RoboDK station: kr30 cnc 072119 dry run.rdk

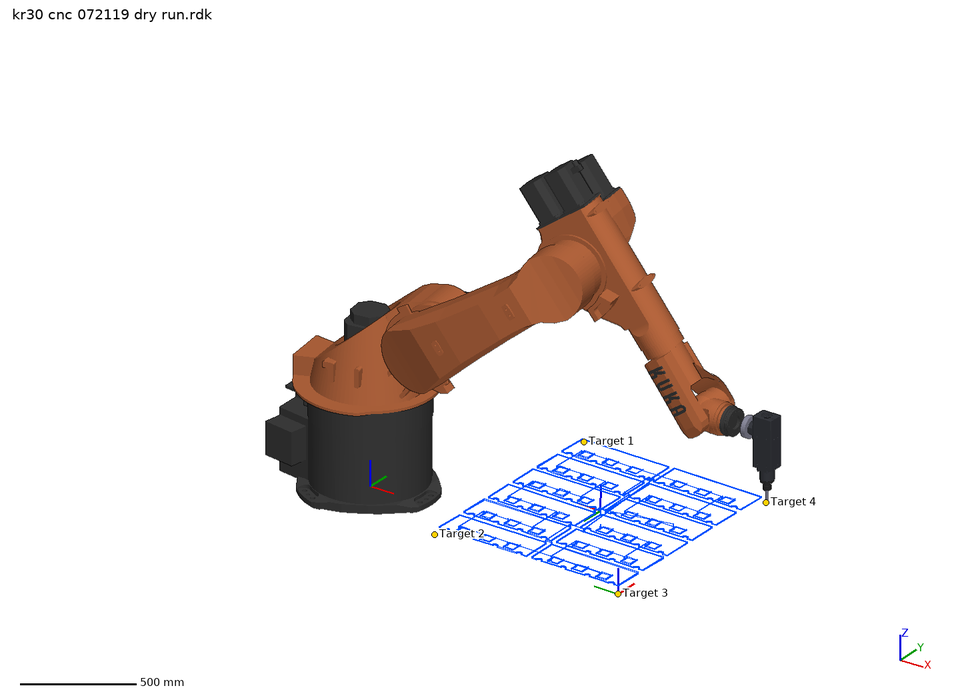
[picture v0: the station drawn from its stored meshes, robots at their saved joint values, targets as dots, program paths as lines]
Station kr30 cnc 072119 dry run. Poses are relative to the parent item; angles as X-Y-Z fixed-axis rotations.
  - frame GIGASHEEN Base at (0, 0, 0) mm
    - robot GIGASHEEN (model KUKA KR 30 HA): 6 axes, payload 30 kg, reach 2033 mm, repeatability 0.05 mm, weight 665 kg
        modified DH rows (alpha deg, a mm, theta deg, d mm): 0, 0, 0, 815; -90, 350, 0, 0; 0, 850, -90, 0; -90, 145, 0, 820; 90, 0, 0, 0; -90, 0, 180, 170
        joint limits [-185, -135, -120, -350, -119, -350] to [185, 35, 158, 350, 119, 350]; home [0, -90, 90, 0, 0, 0]; saved at [-6.898, -35.989, 90.741, -8.88, -55.221, 5.167]
      - tool 1/2" End Mill TCP, TCP at (337.71, -2.2, 160.57) mm, rotated rx 0 ry 90 rz 0 deg, size 415.8 x 102 x 153.6 mm
    - target Target 1 (joint target) at (982.46, 202.21, 406.25) mm, rotated rx -179.95 ry 0.15 rz -89.48 deg; joints [7.49, -59.642, 144.935, 97.969, -90.801, -4.608] of GIGASHEEN
    - target Target 2 (joint target) at (986.83, -921.64, 412.07) mm, rotated rx -179.94 ry 0.15 rz -89.48 deg; joints [51.766, -38.608, 94.384, 136.851, -116.554, -22.567] of GIGASHEEN
    - target Target 3 (joint target) at (1949.02, -919.97, 396.91) mm, rotated rx -179.94 ry 0.14 rz 179.61 deg; joints [29.5, -22.76, 62.288, 41.088, -47.759, -30.404] of GIGASHEEN
    - target Target 4 (joint target) at (1949.02, 190.94, 391.63) mm, rotated rx -179.94 ry 0.14 rz 179.61 deg; joints [-6.898, -35.989, 90.741, -8.88, -55.221, 5.167] of GIGASHEEN
  - machining project Machining Settings: C:/Users/liqui/OneDrive/Desktop/first half pipe jig.apt | rotZ(0) | rotX(0)*rotY(0) | rotZ(0)
  - program Machining (1954 instructions, listed below)
  - program Prog2 (4 instructions, listed below)
  - frame Table at (1949.02, -919.97, 396.91) mm, rotated rx 0.87 ry 0.27 rz 90 deg
    - frame Frame 4 at (550, 480, 40) mm, rotated rx 0 ry 0 rz 90 deg
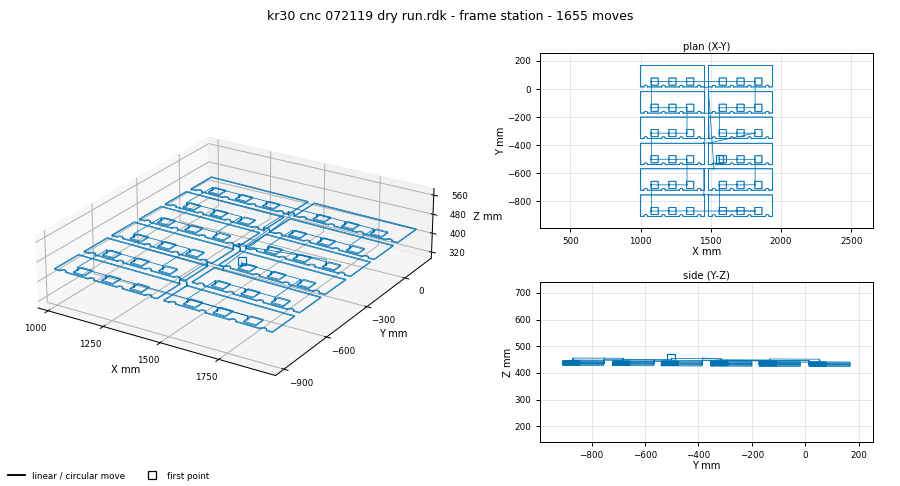
[picture p0: tool path of kr30 cnc 072119 dry run.rdk in frame station, 1655 of 1659 moves have a stored position in this frame; points joined in program order, loops and branches not executed]

--- program Machining (robot GIGASHEEN) ---
  Smooth(0)
  Set Ref.: Frame 4
  Set Tool: 1/2" End Mill TCP
  Show 1/2" End Mill TCP
  Print: /'1001'
  Print: /''
  Print: /'2D Contour2'
  Set speed (500.0 mm/s)
  MoveJ 1 to (-92.16, 131.48, 15) mm, rotated rx 180 ry 0 rz 0 deg; joints [21.909, -52.477, 118.543, 23.9, -67.031, -9.189]
  MoveL 2 to (-92.16, 131.48, 15) mm, rotated rx 180 ry 0 rz 0 deg; joints [21.909, -52.477, 118.543, 23.9, -67.031, -9.189]
  MoveL 3 to (-92.16, 131.48, 15) mm, rotated rx 180 ry 0 rz 0 deg; joints [21.909, -52.477, 118.543, 23.9, -67.031, -9.189]
  Set speed (500.0 mm/s)
  MoveL 4 to (-92.16, 131.48, 6) mm, rotated rx -180 ry 0 rz 0 deg; joints [21.913, -51.95, 118.536, 23.816, -67.508, -8.962]
  Set speed (25.4 mm/s)
  MoveL 5 to (-92.16, 131.48, -3.54) mm, rotated rx 180 ry 0 rz 0 deg; joints [21.917, -51.387, 118.521, 23.73, -68.011, -8.725]
  MoveC 6 to (-91.98, 131.48, -3.99) mm, rotated rx 180 ry 0 rz 0 deg; joints [21.92, -51.367, 118.535, 23.728, -68.042, -8.712] to (-91.53, 131.48, -4.17) mm, rotated rx -180 ry 0 rz 0 deg; joints [21.927, -51.372, 118.57, 23.731, -68.07, -8.702]
  Set speed (50.8 mm/s)
  MoveL 7 to (-90.89, 131.48, -4.18) mm, rotated rx 180 ry 0 rz 0 deg; joints [21.937, -51.395, 118.619, 23.737, -68.095, -8.694]
  MoveC 8 to (-90.44, 131.3, -4.18) mm, rotated rx 180 ry 0 rz 0 deg; joints [21.937, -51.415, 118.66, 23.734, -68.115, -8.685] to (-90.26, 130.85, -4.18) mm, rotated rx -180 ry 0 rz 0 deg; joints [21.922, -51.428, 118.688, 23.715, -68.127, -8.672]
  MoveL 9 to (-90.26, 105.45, -4.17) mm, rotated rx -180 ry 0 rz 0 deg; joints [20.901, -51.776, 119.463, 22.561, -68.365, -8.105]
  MoveL 10 to (-141.06, 105.45, -4.17) mm, rotated rx 180 ry 0 rz 0 deg; joints [20.142, -49.88, 115.443, 22.086, -66.286, -8.677]
  MoveL 11 to (-141.06, 156.25, -4.18) mm, rotated rx 180 ry 0 rz 0 deg; joints [22.112, -49.164, 113.869, 24.362, -65.824, -9.881]
  MoveL 12 to (-90.26, 156.25, -4.18) mm, rotated rx -180 ry 0 rz 0 deg; joints [22.93, -51.06, 117.875, 24.862, -67.882, -9.257]
  MoveL 13 to (-90.26, 130.85, -4.18) mm, rotated rx -180 ry 0 rz 0 deg; joints [21.922, -51.428, 118.688, 23.715, -68.127, -8.672]
  MoveC 14 to (-90.44, 130.4, -4.17) mm, rotated rx 180 ry 0 rz 0 deg; joints [21.901, -51.427, 118.688, 23.693, -68.123, -8.664] to (-90.89, 130.21, -4.18) mm, rotated rx -180 ry 0 rz 0 deg; joints [21.887, -51.413, 118.659, 23.68, -68.107, -8.665]
  MoveL 15 to (-91.53, 130.21, -4.18) mm, rotated rx -180 ry 0 rz 0 deg; joints [21.877, -51.39, 118.609, 23.673, -68.082, -8.673]
  MoveC 16 to (-91.98, 130.21, -3.99) mm, rotated rx 180 ry 0 rz 0 deg; joints [21.869, -51.385, 118.575, 23.67, -68.054, -8.683] to (-92.16, 130.21, -3.54) mm, rotated rx 180 ry 0 rz 0 deg; joints [21.866, -51.404, 118.561, 23.672, -68.023, -8.696]
  Set speed (500.0 mm/s)
  MoveL 17 to (-92.16, 130.21, 5) mm, rotated rx 180 ry 0 rz 0 deg; joints [21.862, -51.909, 118.575, 23.749, -67.573, -8.908]
  MoveL 18 to (-92.16, 131.49, 5) mm, rotated rx -180 ry 0 rz 0 deg; joints [21.913, -51.891, 118.535, 23.807, -67.561, -8.937]
  Set speed (25.4 mm/s)
  MoveL 19 to (-92.16, 131.48, 1.82) mm, rotated rx 180 ry 0 rz 0 deg; joints [21.914, -51.704, 118.531, 23.778, -67.729, -8.858]
  MoveL 20 to (-92.16, 131.48, -7.72) mm, rotated rx 180 ry 0 rz 0 deg; joints [21.919, -51.139, 118.513, 23.693, -68.23, -8.622]
  MoveC 21 to (-91.98, 131.48, -8.16) mm, rotated rx 180 ry 0 rz 0 deg; joints [21.922, -51.119, 118.526, 23.691, -68.261, -8.609] to (-91.53, 131.48, -8.35) mm, rotated rx -180 ry 0 rz 0 deg; joints [21.929, -51.124, 118.56, 23.694, -68.288, -8.599]
  Set speed (50.8 mm/s)
  MoveL 22 to (-90.89, 131.48, -8.35) mm, rotated rx 180 ry 0 rz 0 deg; joints [21.939, -51.148, 118.61, 23.701, -68.314, -8.591]
  MoveC 23 to (-90.44, 131.3, -8.35) mm, rotated rx 180 ry 0 rz 0 deg; joints [21.939, -51.167, 118.651, 23.697, -68.334, -8.582] to (-90.26, 130.85, -8.35) mm, rotated rx -180 ry 0 rz 0 deg; joints [21.924, -51.18, 118.679, 23.679, -68.346, -8.57]
  MoveL 24 to (-90.26, 105.45, -8.35) mm, rotated rx -180 ry 0 rz 0 deg; joints [20.902, -51.526, 119.454, 22.526, -68.588, -8.006]
  MoveL 25 to (-141.06, 105.45, -8.35) mm, rotated rx -180 ry 0 rz 0 deg; joints [20.144, -49.641, 115.434, 22.05, -66.499, -8.584]
  MoveL 26 to (-141.06, 156.25, -8.35) mm, rotated rx 180 ry 0 rz 0 deg; joints [22.114, -48.93, 113.86, 24.322, -66.03, -9.779]
  MoveL 27 to (-90.26, 156.25, -8.35) mm, rotated rx -180 ry 0 rz 0 deg; joints [22.931, -50.815, 117.866, 24.823, -68.097, -9.15]
  MoveL 28 to (-90.26, 130.85, -8.35) mm, rotated rx -180 ry 0 rz 0 deg; joints [21.924, -51.18, 118.679, 23.679, -68.346, -8.57]
  MoveC 29 to (-90.44, 130.4, -8.35) mm, rotated rx 180 ry 0 rz 0 deg; joints [21.903, -51.179, 118.679, 23.657, -68.343, -8.562] to (-90.89, 130.21, -8.35) mm, rotated rx -180 ry 0 rz 0 deg; joints [21.889, -51.165, 118.65, 23.644, -68.326, -8.563]
  MoveL 30 to (-91.53, 130.21, -8.35) mm, rotated rx 180 ry 0 rz 0 deg; joints [21.878, -51.142, 118.6, 23.637, -68.301, -8.57]
  MoveC 31 to (-91.98, 130.21, -8.16) mm, rotated rx -180 ry 0 rz 0 deg; joints [21.871, -51.137, 118.566, 23.634, -68.273, -8.58] to (-92.16, 130.21, -7.72) mm, rotated rx -180 ry 0 rz 0 deg; joints [21.868, -51.157, 118.552, 23.636, -68.242, -8.593]
  Set speed (500.0 mm/s)
  MoveL 32 to (-92.16, 130.21, 6) mm, rotated rx 180 ry 0 rz 0 deg; joints [21.862, -51.968, 118.576, 23.758, -67.52, -8.933]
  MoveL 33 to (-219.16, 131.48, 6) mm, rotated rx -180 ry 0 rz 0 deg; joints [20.042, -46.998, 108.236, 22.771, -62.271, -10.462]
  Set speed (25.4 mm/s)
  MoveL 34 to (-219.16, 131.48, -3.54) mm, rotated rx -180 ry 0 rz 0 deg; joints [20.045, -46.495, 108.222, 22.677, -62.723, -10.251]
  MoveC 35 to (-218.98, 131.48, -3.99) mm, rotated rx -180 ry 0 rz 0 deg; joints [20.048, -46.478, 108.237, 22.673, -62.752, -10.239] to (-218.53, 131.48, -4.17) mm, rotated rx -180 ry 0 rz 0 deg; joints [20.054, -46.487, 108.275, 22.674, -62.78, -10.229]
  Set speed (50.8 mm/s)
  MoveL 36 to (-217.89, 131.49, -4.17) mm, rotated rx -180 ry 0 rz 0 deg; joints [20.063, -46.512, 108.328, 22.678, -62.808, -10.221]
  MoveC 37 to (-217.44, 131.3, -4.18) mm, rotated rx 180 ry 0 rz 0 deg; joints [20.062, -46.533, 108.372, 22.673, -62.829, -10.211] to (-217.26, 130.85, -4.18) mm, rotated rx -180 ry 0 rz 0 deg; joints [20.048, -46.547, 108.402, 22.654, -62.841, -10.197]
  MoveL 38 to (-217.26, 105.45, -4.17) mm, rotated rx 180 ry 0 rz 0 deg; joints [19.099, -46.897, 109.164, 21.526, -63.055, -9.56]
  MoveL 39 to (-268.06, 105.45, -4.17) mm, rotated rx -180 ry 0 rz 0 deg; joints [18.46, -44.806, 104.789, 21.257, -60.816, -10.178]
  MoveL 40 to (-268.06, 156.25, -4.18) mm, rotated rx -180 ry 0 rz 0 deg; joints [20.293, -44.079, 103.221, 23.503, -60.392, -11.532]
  MoveL 41 to (-217.26, 156.25, -4.18) mm, rotated rx -180 ry 0 rz 0 deg; joints [20.986, -46.177, 107.599, 23.778, -62.618, -10.849]
  MoveL 42 to (-217.26, 130.85, -4.18) mm, rotated rx -180 ry 0 rz 0 deg; joints [20.048, -46.547, 108.402, 22.654, -62.841, -10.197]
  MoveC 43 to (-217.44, 130.4, -4.17) mm, rotated rx -180 ry 0 rz 0 deg; joints [20.029, -46.546, 108.4, 22.633, -62.836, -10.188] to (-217.89, 130.21, -4.18) mm, rotated rx -180 ry 0 rz 0 deg; joints [20.016, -46.53, 108.368, 22.622, -62.819, -10.189]
  MoveL 44 to (-218.53, 130.21, -4.18) mm, rotated rx -180 ry 0 rz 0 deg; joints [20.007, -46.505, 108.314, 22.618, -62.791, -10.197]
  MoveC 45 to (-218.98, 130.21, -3.99) mm, rotated rx 180 ry 0 rz 0 deg; joints [20.001, -46.496, 108.276, 22.617, -62.763, -10.206] to (-219.16, 130.21, -3.54) mm, rotated rx -180 ry 0 rz 0 deg; joints [19.998, -46.513, 108.261, 22.62, -62.734, -10.218]
  Set speed (500.0 mm/s)
  MoveL 46 to (-219.16, 130.21, 5) mm, rotated rx -180 ry 0 rz 0 deg; joints [19.995, -46.963, 108.274, 22.704, -62.329, -10.407]
  MoveL 47 to (-219.16, 131.48, 5) mm, rotated rx 180 ry 0 rz 0 deg; joints [20.042, -46.945, 108.235, 22.761, -62.319, -10.44]
  Set speed (25.4 mm/s)
  MoveL 48 to (-219.16, 131.48, 1.82) mm, rotated rx -180 ry 0 rz 0 deg; joints [20.043, -46.778, 108.231, 22.729, -62.469, -10.369]
  MoveL 49 to (-219.16, 131.48, -7.72) mm, rotated rx -180 ry 0 rz 0 deg; joints [20.047, -46.273, 108.214, 22.636, -62.919, -10.159]
  MoveC 50 to (-218.98, 131.48, -8.16) mm, rotated rx -180 ry 0 rz 0 deg; joints [20.05, -46.257, 108.228, 22.633, -62.949, -10.147] to (-218.53, 131.48, -8.35) mm, rotated rx -180 ry 0 rz 0 deg; joints [20.056, -46.265, 108.266, 22.634, -62.977, -10.138]
  Set speed (50.8 mm/s)
  MoveL 51 to (-217.89, 131.48, -8.35) mm, rotated rx -180 ry 0 rz 0 deg; joints [20.064, -46.291, 108.32, 22.638, -63.004, -10.13]
  MoveC 52 to (-217.44, 131.3, -8.35) mm, rotated rx -180 ry 0 rz 0 deg; joints [20.064, -46.311, 108.363, 22.633, -63.025, -10.119] to (-217.26, 130.85, -8.35) mm, rotated rx 180 ry 0 rz 0 deg; joints [20.05, -46.325, 108.393, 22.614, -63.037, -10.106]
  MoveL 53 to (-217.26, 105.45, -8.35) mm, rotated rx -180 ry 0 rz 0 deg; joints [19.101, -46.674, 109.156, 21.488, -63.255, -9.473]
  MoveL 54 to (-268.06, 105.45, -8.35) mm, rotated rx -180 ry 0 rz 0 deg; joints [18.461, -44.592, 104.78, 21.217, -61.008, -10.094]
  MoveL 55 to (-268.06, 156.25, -8.35) mm, rotated rx -180 ry 0 rz 0 deg; joints [20.295, -43.868, 103.212, 23.459, -60.578, -11.44]
  MoveL 56 to (-217.26, 156.25, -8.35) mm, rotated rx 180 ry 0 rz 0 deg; joints [20.987, -45.957, 107.59, 23.736, -62.812, -10.754]
  MoveL 57 to (-217.26, 130.85, -8.35) mm, rotated rx 180 ry 0 rz 0 deg; joints [20.05, -46.325, 108.393, 22.614, -63.037, -10.106]
  MoveC 58 to (-217.44, 130.4, -8.35) mm, rotated rx 180 ry 0 rz 0 deg; joints [20.03, -46.324, 108.391, 22.593, -63.033, -10.097] to (-217.89, 130.21, -8.35) mm, rotated rx -180 ry 0 rz 0 deg; joints [20.017, -46.309, 108.359, 22.582, -63.015, -10.098]
  MoveL 59 to (-218.53, 130.21, -8.35) mm, rotated rx -180 ry 0 rz 0 deg; joints [20.009, -46.283, 108.305, 22.578, -62.988, -10.106]
  MoveC 60 to (-218.98, 130.21, -8.16) mm, rotated rx 180 ry 0 rz 0 deg; joints [20.003, -46.275, 108.267, 22.577, -62.96, -10.115] to (-219.16, 130.22, -7.72) mm, rotated rx -180 ry 0 rz 0 deg; joints [20, -46.291, 108.253, 22.58, -62.93, -10.127]
  Set speed (500.0 mm/s)
  MoveL 61 to (-219.16, 130.21, 6) mm, rotated rx -180 ry 0 rz 0 deg; joints [19.995, -47.016, 108.276, 22.714, -62.282, -10.429]
  MoveL 62 to (-346.16, 131.48, 6) mm, rotated rx -180 ry 0 rz 0 deg; joints [18.455, -41.516, 96.931, 22.283, -56.572, -12.158]
  Set speed (25.4 mm/s)
  MoveL 63 to (-346.16, 131.48, -3.54) mm, rotated rx 180 ry 0 rz 0 deg; joints [18.458, -41.062, 96.917, 22.178, -56.98, -11.961]
  MoveC 64 to (-345.98, 131.48, -3.99) mm, rotated rx -180 ry 0 rz 0 deg; joints [18.461, -41.049, 96.933, 22.173, -57.008, -11.95] to (-345.53, 131.48, -4.17) mm, rotated rx -180 ry 0 rz 0 deg; joints [18.466, -41.06, 96.975, 22.172, -57.037, -11.939]
  Set speed (50.8 mm/s)
  MoveL 65 to (-344.89, 131.48, -4.17) mm, rotated rx -180 ry 0 rz 0 deg; joints [18.473, -41.089, 97.035, 22.173, -57.067, -11.93]
  MoveC 66 to (-344.44, 131.3, -4.17) mm, rotated rx 180 ry 0 rz 0 deg; joints [18.472, -41.112, 97.083, 22.165, -57.09, -11.918] to (-344.26, 130.85, -4.18) mm, rotated rx -180 ry 0 rz 0 deg; joints [18.459, -41.127, 97.114, 22.146, -57.103, -11.902]
  MoveL 67 to (-344.26, 105.45, -4.17) mm, rotated rx -180 ry 0 rz 0 deg; joints [17.574, -41.489, 97.887, 21.018, -57.305, -11.178]
  MoveL 68 to (-395.06, 105.45, -4.18) mm, rotated rx -180 ry 0 rz 0 deg; joints [17.029, -39.137, 93.017, 20.982, -54.842, -11.914]
  MoveL 69 to (-395.06, 156.25, -4.17) mm, rotated rx -180 ry 0 rz 0 deg; joints [18.741, -38.377, 91.402, 23.257, -54.433, -13.468]
  MoveL 70 to (-344.26, 156.25, -4.18) mm, rotated rx 180 ry 0 rz 0 deg; joints [19.334, -40.745, 96.299, 23.273, -56.893, -12.643]
  MoveL 71 to (-344.26, 130.85, -4.18) mm, rotated rx -180 ry 0 rz 0 deg; joints [18.459, -41.127, 97.114, 22.146, -57.103, -11.902]
  MoveC 72 to (-344.44, 130.4, -4.18) mm, rotated rx -180 ry 0 rz 0 deg; joints [18.441, -41.125, 97.111, 22.125, -57.097, -11.892] to (-344.89, 130.22, -4.18) mm, rotated rx -180 ry 0 rz 0 deg; joints [18.429, -41.108, 97.074, 22.116, -57.078, -11.893]
  MoveL 73 to (-345.53, 130.21, -4.18) mm, rotated rx 180 ry 0 rz 0 deg; joints [18.422, -41.079, 97.015, 22.115, -57.048, -11.902]
  MoveC 74 to (-345.98, 130.21, -3.99) mm, rotated rx -180 ry 0 rz 0 deg; joints [18.417, -41.068, 96.973, 22.117, -57.018, -11.913] to (-346.16, 130.21, -3.54) mm, rotated rx 180 ry 0 rz 0 deg; joints [18.414, -41.081, 96.956, 22.121, -56.99, -11.925]
  Set speed (500.0 mm/s)
  MoveL 75 to (-346.16, 130.21, 5) mm, rotated rx -180 ry 0 rz 0 deg; joints [18.411, -41.488, 96.969, 22.215, -56.625, -12.101]
  MoveL 76 to (-346.16, 131.48, 5) mm, rotated rx -180 ry 0 rz 0 deg; joints [18.455, -41.469, 96.93, 22.272, -56.615, -12.138]
  Set speed (25.4 mm/s)
  MoveL 77 to (-346.16, 131.48, 1.82) mm, rotated rx -180 ry 0 rz 0 deg; joints [18.456, -41.318, 96.926, 22.236, -56.751, -12.072]
  MoveL 78 to (-346.16, 131.48, -7.72) mm, rotated rx -180 ry 0 rz 0 deg; joints [18.46, -40.862, 96.908, 22.133, -57.158, -11.876]
  MoveC 79 to (-345.98, 131.48, -8.16) mm, rotated rx 180 ry 0 rz 0 deg; joints [18.462, -40.849, 96.925, 22.128, -57.186, -11.865] to (-345.53, 131.48, -8.35) mm, rotated rx -180 ry 0 rz 0 deg; joints [18.467, -40.86, 96.966, 22.127, -57.215, -11.854]
  Set speed (50.8 mm/s)
  MoveL 80 to (-344.89, 131.48, -8.35) mm, rotated rx -180 ry 0 rz 0 deg; joints [18.475, -40.889, 97.026, 22.128, -57.245, -11.845]
  MoveC 81 to (-344.44, 131.3, -8.35) mm, rotated rx 180 ry 0 rz 0 deg; joints [18.473, -40.912, 97.074, 22.12, -57.268, -11.833] to (-344.26, 130.85, -8.35) mm, rotated rx -180 ry 0 rz 0 deg; joints [18.46, -40.927, 97.105, 22.101, -57.28, -11.817]
  MoveL 82 to (-344.26, 105.45, -8.35) mm, rotated rx 180 ry 0 rz 0 deg; joints [17.576, -41.287, 97.879, 20.976, -57.485, -11.097]
  MoveL 83 to (-395.06, 105.45, -8.35) mm, rotated rx -180 ry 0 rz 0 deg; joints [17.03, -38.943, 93.009, 20.937, -55.015, -11.834]
  MoveL 84 to (-395.06, 156.25, -8.35) mm, rotated rx -180 ry 0 rz 0 deg; joints [18.742, -38.186, 91.393, 23.207, -54.602, -13.38]
  MoveL 85 to (-344.26, 156.25, -8.35) mm, rotated rx -180 ry 0 rz 0 deg; joints [19.335, -40.546, 96.29, 23.226, -57.068, -12.555]
  MoveL 86 to (-344.26, 130.85, -8.35) mm, rotated rx -180 ry 0 rz 0 deg; joints [18.46, -40.927, 97.105, 22.101, -57.28, -11.817]
  MoveC 87 to (-344.44, 130.4, -8.35) mm, rotated rx -180 ry 0 rz 0 deg; joints [18.442, -40.925, 97.102, 22.081, -57.275, -11.807] to (-344.89, 130.21, -8.35) mm, rotated rx -180 ry 0 rz 0 deg; joints [18.431, -40.908, 97.066, 22.072, -57.255, -11.808]
  MoveL 88 to (-345.53, 130.21, -8.35) mm, rotated rx -180 ry 0 rz 0 deg; joints [18.423, -40.879, 97.006, 22.071, -57.225, -11.818]
  MoveC 89 to (-345.98, 130.21, -8.16) mm, rotated rx -180 ry 0 rz 0 deg; joints [18.418, -40.868, 96.964, 22.072, -57.196, -11.828] to (-346.16, 130.21, -7.72) mm, rotated rx 180 ry 0 rz 0 deg; joints [18.416, -40.881, 96.948, 22.076, -57.168, -11.84]
  Set speed (500.0 mm/s)
  MoveL 90 to (-346.16, 130.21, 6) mm, rotated rx -180 ry 0 rz 0 deg; joints [18.411, -41.535, 96.971, 22.226, -56.582, -12.121]
  MoveL 91 to (-346.16, 313.35, 6) mm, rotated rx 180 ry 0 rz 0 deg; joints [24.501, -38.28, 90.113, 30.424, -54.956, -17.966]
  Set speed (25.4 mm/s)
  MoveL 92 to (-346.16, 313.35, -3.54) mm, rotated rx 180 ry 0 rz 0 deg; joints [24.504, -37.849, 90.099, 30.281, -55.317, -17.711]
  MoveC 93 to (-345.98, 313.35, -3.99) mm, rotated rx -180 ry 0 rz 0 deg; joints [24.507, -37.837, 90.116, 30.275, -55.343, -17.695] to (-345.53, 313.35, -4.17) mm, rotated rx -180 ry 0 rz 0 deg; joints [24.514, -37.85, 90.159, 30.272, -55.371, -17.681]
  Set speed (50.8 mm/s)
  MoveL 94 to (-344.89, 313.36, -4.18) mm, rotated rx -180 ry 0 rz 0 deg; joints [24.523, -37.879, 90.22, 30.271, -55.401, -17.668]
  MoveC 95 to (-344.44, 313.17, -4.18) mm, rotated rx -180 ry 0 rz 0 deg; joints [24.524, -37.904, 90.271, 30.263, -55.424, -17.652] to (-344.26, 312.72, -4.18) mm, rotated rx -180 ry 0 rz 0 deg; joints [24.512, -37.922, 90.309, 30.243, -55.438, -17.633]
  MoveL 96 to (-344.26, 287.32, -4.18) mm, rotated rx -180 ry 0 rz 0 deg; joints [23.697, -38.438, 91.398, 29.106, -55.691, -16.768]
  MoveL 97 to (-395.06, 287.32, -4.18) mm, rotated rx 180 ry 0 rz 0 deg; joints [22.998, -36.008, 86.396, 29.181, -53.234, -17.841]
  MoveL 98 to (-395.06, 338.12, -4.18) mm, rotated rx 180 ry 0 rz 0 deg; joints [24.581, -34.921, 84.111, 31.512, -52.717, -19.704]
  MoveL 99 to (-344.26, 338.12, -4.18) mm, rotated rx 180 ry 0 rz 0 deg; joints [25.316, -37.384, 89.172, 31.383, -55.178, -18.521]
  MoveL 100 to (-344.26, 312.72, -4.17) mm, rotated rx 180 ry 0 rz 0 deg; joints [24.512, -37.922, 90.309, 30.243, -55.438, -17.633]
  MoveC 101 to (-344.44, 312.27, -4.17) mm, rotated rx -180 ry 0 rz 0 deg; joints [24.495, -37.923, 90.31, 30.223, -55.433, -17.621] to (-344.89, 312.08, -4.17) mm, rotated rx -180 ry 0 rz 0 deg; joints [24.483, -37.906, 90.275, 30.214, -55.414, -17.624]
  MoveL 102 to (-345.53, 312.08, -4.18) mm, rotated rx 180 ry 0 rz 0 deg; joints [24.473, -37.876, 90.214, 30.215, -55.384, -17.637]
  MoveC 103 to (-345.98, 312.08, -3.99) mm, rotated rx 180 ry 0 rz 0 deg; joints [24.467, -37.864, 90.171, 30.218, -55.356, -17.652] to (-346.16, 312.08, -3.54) mm, rotated rx 180 ry 0 rz 0 deg; joints [24.464, -37.875, 90.154, 30.224, -55.33, -17.667]
  Set speed (500.0 mm/s)
  MoveL 104 to (-346.16, 312.08, 5) mm, rotated rx -180 ry 0 rz 0 deg; joints [24.461, -38.262, 90.167, 30.352, -55.007, -17.895]
  MoveL 105 to (-346.16, 313.35, 5) mm, rotated rx -180 ry 0 rz 0 deg; joints [24.501, -38.235, 90.112, 30.409, -54.994, -17.939]
  Set speed (25.4 mm/s)
  MoveL 106 to (-346.16, 313.35, 1.82) mm, rotated rx -180 ry 0 rz 0 deg; joints [24.502, -38.092, 90.108, 30.361, -55.115, -17.854]
  MoveL 107 to (-346.16, 313.35, -7.71) mm, rotated rx -180 ry 0 rz 0 deg; joints [24.506, -37.659, 90.09, 30.22, -55.474, -17.601]
  MoveC 108 to (-345.98, 313.35, -8.16) mm, rotated rx 180 ry 0 rz 0 deg; joints [24.509, -37.647, 90.107, 30.213, -55.5, -17.586] to (-345.53, 313.35, -8.35) mm, rotated rx -180 ry 0 rz 0 deg; joints [24.515, -37.66, 90.15, 30.211, -55.528, -17.571]
  Set speed (50.8 mm/s)
  MoveL 109 to (-344.89, 313.35, -8.35) mm, rotated rx 180 ry 0 rz 0 deg; joints [24.525, -37.689, 90.211, 30.21, -55.558, -17.558]
  MoveC 110 to (-344.44, 313.17, -8.35) mm, rotated rx -180 ry 0 rz 0 deg; joints [24.525, -37.714, 90.262, 30.202, -55.582, -17.542] to (-344.26, 312.72, -8.35) mm, rotated rx -180 ry 0 rz 0 deg; joints [24.514, -37.732, 90.3, 30.182, -55.595, -17.523]
  MoveL 111 to (-344.26, 287.32, -8.35) mm, rotated rx -180 ry 0 rz 0 deg; joints [23.699, -38.246, 91.389, 29.047, -55.852, -16.661]
  MoveL 112 to (-395.06, 287.32, -8.35) mm, rotated rx 180 ry 0 rz 0 deg; joints [22.999, -35.823, 86.387, 29.119, -53.388, -17.735]
  MoveL 113 to (-395.06, 338.12, -8.35) mm, rotated rx -180 ry 0 rz 0 deg; joints [24.583, -34.738, 84.102, 31.445, -52.865, -19.591]
  MoveL 114 to (-344.26, 338.12, -8.35) mm, rotated rx 180 ry 0 rz 0 deg; joints [25.318, -37.195, 89.164, 31.32, -55.332, -18.408]
  MoveL 115 to (-344.26, 312.72, -8.35) mm, rotated rx -180 ry 0 rz 0 deg; joints [24.514, -37.732, 90.3, 30.182, -55.595, -17.523]
  MoveC 116 to (-344.44, 312.27, -8.35) mm, rotated rx 180 ry 0 rz 0 deg; joints [24.497, -37.733, 90.302, 30.162, -55.591, -17.511] to (-344.89, 312.08, -8.35) mm, rotated rx -180 ry 0 rz 0 deg; joints [24.484, -37.716, 90.267, 30.153, -55.571, -17.514]
  MoveL 117 to (-345.53, 312.08, -8.35) mm, rotated rx 180 ry 0 rz 0 deg; joints [24.475, -37.686, 90.205, 30.154, -55.541, -17.528]
  MoveC 118 to (-345.98, 312.08, -8.16) mm, rotated rx 180 ry 0 rz 0 deg; joints [24.468, -37.674, 90.163, 30.157, -55.513, -17.542] to (-346.16, 312.08, -7.72) mm, rotated rx 180 ry 0 rz 0 deg; joints [24.465, -37.685, 90.146, 30.163, -55.487, -17.558]
  Set speed (500.0 mm/s)
  MoveL 119 to (-346.16, 312.08, 6) mm, rotated rx 180 ry 0 rz 0 deg; joints [24.46, -38.307, 90.168, 30.367, -54.969, -17.921]
  MoveL 120 to (-219.16, 313.35, 6) mm, rotated rx -180 ry 0 rz 0 deg; joints [26.482, -43.877, 101.587, 30.778, -60.597, -15.594]
  Set speed (25.4 mm/s)
  MoveL 121 to (-219.16, 313.35, -3.54) mm, rotated rx 180 ry 0 rz 0 deg; joints [26.486, -43.405, 101.574, 30.651, -60.993, -15.327]
  MoveC 122 to (-218.98, 313.35, -3.99) mm, rotated rx -180 ry 0 rz 0 deg; joints [26.489, -43.39, 101.589, 30.646, -61.019, -15.312] to (-218.53, 313.35, -4.17) mm, rotated rx -180 ry 0 rz 0 deg; joints [26.496, -43.399, 101.626, 30.647, -61.046, -15.299]
  Set speed (50.8 mm/s)
  MoveL 123 to (-217.89, 313.35, -4.17) mm, rotated rx -180 ry 0 rz 0 deg; joints [26.507, -43.425, 101.68, 30.65, -61.073, -15.288]
  MoveC 124 to (-217.44, 313.17, -4.17) mm, rotated rx -180 ry 0 rz 0 deg; joints [26.508, -43.448, 101.726, 30.645, -61.094, -15.275] to (-217.26, 312.72, -4.18) mm, rotated rx -180 ry 0 rz 0 deg; joints [26.496, -43.464, 101.761, 30.627, -61.106, -15.258]
  MoveL 125 to (-217.26, 287.32, -4.18) mm, rotated rx 180 ry 0 rz 0 deg; joints [25.634, -43.956, 102.815, 29.523, -61.366, -14.493]
  MoveL 126 to (-268.06, 287.32, -4.18) mm, rotated rx 180 ry 0 rz 0 deg; joints [24.825, -41.833, 98.411, 29.263, -59.167, -15.349]
  MoveL 127 to (-268.06, 338.12, -4.17) mm, rotated rx -180 ry 0 rz 0 deg; joints [26.499, -40.813, 96.241, 31.488, -58.649, -16.97]
  MoveL 128 to (-217.26, 338.12, -4.17) mm, rotated rx -180 ry 0 rz 0 deg; joints [27.346, -42.951, 100.666, 31.729, -60.841, -16.044]
  MoveL 129 to (-217.26, 312.72, -4.18) mm, rotated rx -180 ry 0 rz 0 deg; joints [26.496, -43.464, 101.761, 30.627, -61.106, -15.258]
  MoveC 130 to (-217.44, 312.27, -4.17) mm, rotated rx 180 ry 0 rz 0 deg; joints [26.478, -43.465, 101.764, 30.606, -61.103, -15.248] to (-217.89, 312.08, -4.18) mm, rotated rx -180 ry 0 rz 0 deg; joints [26.464, -43.451, 101.734, 30.595, -61.086, -15.25]
  MoveL 131 to (-218.53, 312.08, -4.17) mm, rotated rx -180 ry 0 rz 0 deg; joints [26.454, -43.425, 101.68, 30.591, -61.059, -15.26]
  MoveC 132 to (-218.98, 312.08, -3.99) mm, rotated rx -180 ry 0 rz 0 deg; joints [26.446, -43.415, 101.642, 30.591, -61.032, -15.273] to (-219.16, 312.08, -3.54) mm, rotated rx -180 ry 0 rz 0 deg; joints [26.443, -43.43, 101.627, 30.596, -61.006, -15.289]
  Set speed (500.0 mm/s)
  MoveL 133 to (-219.16, 312.08, 5) mm, rotated rx 180 ry 0 rz 0 deg; joints [26.439, -43.853, 101.64, 30.709, -60.652, -15.526]
  MoveL 134 to (-219.16, 313.35, 5) mm, rotated rx 180 ry 0 rz 0 deg; joints [26.482, -43.828, 101.586, 30.764, -60.639, -15.566]
  Set speed (25.4 mm/s)
  MoveL 135 to (-219.16, 313.35, 1.82) mm, rotated rx -180 ry 0 rz 0 deg; joints [26.483, -43.671, 101.582, 30.722, -60.771, -15.477]
  MoveL 136 to (-219.16, 313.36, -7.72) mm, rotated rx -180 ry 0 rz 0 deg; joints [26.487, -43.197, 101.565, 30.597, -61.165, -15.212]
  MoveC 137 to (-218.98, 313.35, -8.16) mm, rotated rx 180 ry 0 rz 0 deg; joints [26.491, -43.182, 101.58, 30.592, -61.191, -15.197] to (-218.53, 313.36, -8.35) mm, rotated rx -180 ry 0 rz 0 deg; joints [26.498, -43.191, 101.618, 30.593, -61.218, -15.184]
  Set speed (50.8 mm/s)
  MoveL 138 to (-217.89, 313.35, -8.35) mm, rotated rx 180 ry 0 rz 0 deg; joints [26.509, -43.217, 101.672, 30.596, -61.245, -15.173]
  MoveC 139 to (-217.44, 313.17, -8.35) mm, rotated rx -180 ry 0 rz 0 deg; joints [26.51, -43.239, 101.718, 30.591, -61.266, -15.16] to (-217.26, 312.72, -8.35) mm, rotated rx 180 ry 0 rz 0 deg; joints [26.498, -43.256, 101.753, 30.573, -61.278, -15.143]
  MoveL 140 to (-217.26, 287.32, -8.35) mm, rotated rx -180 ry 0 rz 0 deg; joints [25.636, -43.746, 102.806, 29.471, -61.542, -14.381]
  MoveL 141 to (-268.06, 287.32, -8.35) mm, rotated rx -180 ry 0 rz 0 deg; joints [24.826, -41.63, 98.402, 29.208, -59.337, -15.239]
  MoveL 142 to (-268.06, 338.12, -8.35) mm, rotated rx 180 ry 0 rz 0 deg; joints [26.501, -40.614, 96.233, 31.43, -58.812, -16.855]
  MoveL 143 to (-217.26, 338.12, -8.35) mm, rotated rx -180 ry 0 rz 0 deg; joints [27.348, -42.745, 100.657, 31.673, -61.009, -15.926]
  MoveL 144 to (-217.26, 312.72, -8.35) mm, rotated rx 180 ry 0 rz 0 deg; joints [26.498, -43.256, 101.753, 30.573, -61.278, -15.143]
  MoveC 145 to (-217.44, 312.27, -8.35) mm, rotated rx -180 ry 0 rz 0 deg; joints [26.48, -43.257, 101.756, 30.552, -61.275, -15.133] to (-217.89, 312.08, -8.35) mm, rotated rx -180 ry 0 rz 0 deg; joints [26.466, -43.242, 101.725, 30.541, -61.258, -15.135]
  MoveL 146 to (-218.53, 312.08, -8.35) mm, rotated rx -180 ry 0 rz 0 deg; joints [26.455, -43.216, 101.671, 30.537, -61.231, -15.145]
  MoveC 147 to (-218.98, 312.08, -8.16) mm, rotated rx 180 ry 0 rz 0 deg; joints [26.448, -43.207, 101.634, 30.537, -61.204, -15.158] to (-219.16, 312.08, -7.72) mm, rotated rx -180 ry 0 rz 0 deg; joints [26.445, -43.222, 101.619, 30.542, -61.178, -15.174]
  Set speed (500.0 mm/s)
  MoveL 148 to (-219.16, 312.08, 6) mm, rotated rx -180 ry 0 rz 0 deg; joints [26.439, -43.903, 101.641, 30.722, -60.61, -15.554]
  MoveL 149 to (-92.16, 313.35, 6) mm, rotated rx -180 ry 0 rz 0 deg; joints [28.782, -48.856, 111.85, 31.879, -65.703, -13.605]
  Set speed (25.4 mm/s)
  MoveL 150 to (-92.16, 313.35, -3.54) mm, rotated rx 180 ry 0 rz 0 deg; joints [28.786, -48.334, 111.836, 31.764, -66.135, -13.313]
  MoveC 151 to (-91.98, 313.35, -3.99) mm, rotated rx -180 ry 0 rz 0 deg; joints [28.79, -48.316, 111.85, 31.761, -66.163, -13.297] to (-91.53, 313.35, -4.17) mm, rotated rx -180 ry 0 rz 0 deg; joints [28.799, -48.322, 111.884, 31.764, -66.189, -13.285]
  Set speed (50.8 mm/s)
  MoveL 152 to (-90.89, 313.35, -4.18) mm, rotated rx -180 ry 0 rz 0 deg; joints [28.811, -48.346, 111.933, 31.771, -66.213, -13.275]
  MoveC 153 to (-90.44, 313.17, -4.18) mm, rotated rx -180 ry 0 rz 0 deg; joints [28.813, -48.366, 111.975, 31.769, -66.233, -13.263] to (-90.26, 312.72, -4.18) mm, rotated rx -180 ry 0 rz 0 deg; joints [28.801, -48.381, 112.008, 31.751, -66.245, -13.248]
  MoveL 154 to (-90.26, 287.32, -4.17) mm, rotated rx -180 ry 0 rz 0 deg; joints [27.888, -48.865, 113.06, 30.652, -66.523, -12.552]
  MoveL 155 to (-141.06, 287.32, -4.18) mm, rotated rx 180 ry 0 rz 0 deg; joints [26.944, -46.965, 109.081, 30.121, -64.514, -13.303]
  MoveL 156 to (-141.06, 338.12, -4.18) mm, rotated rx -180 ry 0 rz 0 deg; joints [28.715, -45.973, 106.942, 32.313, -63.97, -14.764]
  MoveL 157 to (-90.26, 338.12, -4.17) mm, rotated rx 180 ry 0 rz 0 deg; joints [29.698, -47.878, 110.917, 32.843, -65.963, -13.964]
  MoveL 158 to (-90.26, 312.72, -4.18) mm, rotated rx -180 ry 0 rz 0 deg; joints [28.801, -48.381, 112.008, 31.751, -66.245, -13.248]
  MoveC 159 to (-90.44, 312.27, -4.18) mm, rotated rx 180 ry 0 rz 0 deg; joints [28.781, -48.383, 112.013, 31.73, -66.243, -13.238] to (-90.89, 312.08, -4.17) mm, rotated rx 180 ry 0 rz 0 deg; joints [28.766, -48.37, 111.986, 31.717, -66.227, -13.24]
  MoveL 160 to (-91.53, 312.08, -4.18) mm, rotated rx -180 ry 0 rz 0 deg; joints [28.753, -48.347, 111.937, 31.709, -66.203, -13.249]
  MoveC 161 to (-91.98, 312.08, -3.99) mm, rotated rx -180 ry 0 rz 0 deg; joints [28.745, -48.341, 111.903, 31.706, -66.177, -13.262] to (-92.16, 312.08, -3.54) mm, rotated rx -180 ry 0 rz 0 deg; joints [28.741, -48.358, 111.89, 31.71, -66.149, -13.278]
  Set speed (500.0 mm/s)
  MoveL 162 to (-92.16, 312.08, 5) mm, rotated rx 180 ry 0 rz 0 deg; joints [28.737, -48.826, 111.903, 31.812, -65.762, -13.538]
  MoveL 163 to (-92.16, 313.36, 5) mm, rotated rx -180 ry 0 rz 0 deg; joints [28.782, -48.801, 111.849, 31.867, -65.748, -13.574]
  Set speed (25.4 mm/s)
  MoveL 164 to (-92.16, 313.35, 1.83) mm, rotated rx -180 ry 0 rz 0 deg; joints [28.783, -48.628, 111.845, 31.829, -65.892, -13.477]
  MoveL 165 to (-92.16, 313.35, -7.71) mm, rotated rx 180 ry 0 rz 0 deg; joints [28.788, -48.104, 111.828, 31.715, -66.324, -13.187]
  MoveC 166 to (-91.98, 313.35, -8.16) mm, rotated rx 180 ry 0 rz 0 deg; joints [28.792, -48.086, 111.841, 31.712, -66.351, -13.171] to (-91.53, 313.35, -8.35) mm, rotated rx -180 ry 0 rz 0 deg; joints [28.801, -48.093, 111.875, 31.715, -66.377, -13.158]
  Set speed (50.8 mm/s)
  MoveL 167 to (-90.89, 313.35, -8.35) mm, rotated rx 180 ry 0 rz 0 deg; joints [28.813, -48.116, 111.924, 31.722, -66.402, -13.149]
  MoveC 168 to (-90.44, 313.17, -8.35) mm, rotated rx -180 ry 0 rz 0 deg; joints [28.815, -48.136, 111.966, 31.72, -66.421, -13.137] to (-90.26, 312.72, -8.35) mm, rotated rx -180 ry 0 rz 0 deg; joints [28.803, -48.151, 111.999, 31.702, -66.433, -13.122]
  MoveL 169 to (-90.26, 287.32, -8.35) mm, rotated rx 180 ry 0 rz 0 deg; joints [27.89, -48.633, 113.052, 30.605, -66.716, -12.428]
  MoveL 170 to (-141.06, 287.32, -8.35) mm, rotated rx 180 ry 0 rz 0 deg; joints [26.946, -46.741, 109.072, 30.072, -64.7, -13.185]
  MoveL 171 to (-141.06, 338.12, -8.35) mm, rotated rx -180 ry 0 rz 0 deg; joints [28.716, -45.754, 106.933, 32.261, -64.148, -14.64]
  MoveL 172 to (-90.26, 338.12, -8.35) mm, rotated rx -180 ry 0 rz 0 deg; joints [29.7, -47.65, 110.908, 32.793, -66.147, -13.835]
  MoveL 173 to (-90.26, 312.72, -8.35) mm, rotated rx -180 ry 0 rz 0 deg; joints [28.803, -48.151, 111.999, 31.702, -66.433, -13.122]
  MoveC 174 to (-90.44, 312.27, -8.35) mm, rotated rx -180 ry 0 rz 0 deg; joints [28.783, -48.153, 112.004, 31.681, -66.431, -13.112] to (-90.89, 312.08, -8.35) mm, rotated rx 180 ry 0 rz 0 deg; joints [28.768, -48.14, 111.977, 31.668, -66.416, -13.114]
  MoveL 175 to (-91.53, 312.08, -8.35) mm, rotated rx -180 ry 0 rz 0 deg; joints [28.755, -48.117, 111.929, 31.66, -66.391, -13.123]
  MoveC 176 to (-91.98, 312.08, -8.16) mm, rotated rx -180 ry 0 rz 0 deg; joints [28.747, -48.111, 111.895, 31.658, -66.365, -13.136] to (-92.16, 312.08, -7.72) mm, rotated rx -180 ry 0 rz 0 deg; joints [28.743, -48.129, 111.881, 31.661, -66.338, -13.152]
  Set speed (500.0 mm/s)
  MoveL 177 to (-92.16, 312.08, 6) mm, rotated rx -180 ry 0 rz 0 deg; joints [28.736, -48.881, 111.904, 31.824, -65.716, -13.569]
  MoveL 178 to (-92.16, 499.69, 6) mm, rotated rx 180 ry 0 rz 0 deg; joints [34.993, -44.649, 102.911, 39.778, -63.653, -19.397]
  Set speed (25.4 mm/s)
  MoveL 179 to (-92.16, 499.69, -3.54) mm, rotated rx 180 ry 0 rz 0 deg; joints [34.998, -44.171, 102.898, 39.637, -64.012, -19.069]
  MoveC 180 to (-91.98, 499.69, -3.99) mm, rotated rx 180 ry 0 rz 0 deg; joints [35.002, -44.155, 102.911, 39.633, -64.036, -19.05] to (-91.53, 499.69, -4.17) mm, rotated rx -180 ry 0 rz 0 deg; joints [35.012, -44.162, 102.946, 39.635, -64.06, -19.035]
  Set speed (50.8 mm/s)
  MoveL 181 to (-90.89, 499.69, -4.18) mm, rotated rx 180 ry 0 rz 0 deg; joints [35.026, -44.186, 102.995, 39.641, -64.084, -19.024]
  MoveC 182 to (-90.44, 499.51, -4.17) mm, rotated rx -180 ry 0 rz 0 deg; joints [35.03, -44.208, 103.039, 39.638, -64.103, -19.009] to (-90.26, 499.06, -4.18) mm, rotated rx 180 ry 0 rz 0 deg; joints [35.02, -44.226, 103.078, 39.622, -64.115, -18.99]
  MoveL 183 to (-90.26, 473.66, -4.18) mm, rotated rx 180 ry 0 rz 0 deg; joints [34.221, -44.857, 104.424, 38.566, -64.412, -18.138]
  MoveL 184 to (-141.06, 473.66, -4.17) mm, rotated rx -180 ry 0 rz 0 deg; joints [33.155, -42.929, 100.434, 38.077, -62.45, -19.078]
  MoveL 185 to (-141.06, 524.46, -4.18) mm, rotated rx -180 ry 0 rz 0 deg; joints [34.714, -41.63, 97.681, 40.216, -61.861, -20.866]
  MoveL 186 to (-90.26, 524.46, -4.17) mm, rotated rx -180 ry 0 rz 0 deg; joints [35.803, -43.573, 101.689, 40.674, -63.816, -19.867]
  MoveL 187 to (-90.26, 499.06, -4.18) mm, rotated rx 180 ry 0 rz 0 deg; joints [35.02, -44.226, 103.078, 39.622, -64.115, -18.99]
  MoveC 188 to (-90.44, 498.61, -4.17) mm, rotated rx -180 ry 0 rz 0 deg; joints [35.002, -44.23, 103.087, 39.601, -64.113, -18.978] to (-90.89, 498.42, -4.17) mm, rotated rx -180 ry 0 rz 0 deg; joints [34.986, -44.218, 103.063, 39.589, -64.098, -18.98]
  MoveL 189 to (-91.53, 498.42, -4.17) mm, rotated rx -180 ry 0 rz 0 deg; joints [34.972, -44.195, 103.014, 39.582, -64.074, -18.992]
  MoveC 190 to (-91.98, 498.42, -3.99) mm, rotated rx -180 ry 0 rz 0 deg; joints [34.963, -44.187, 102.98, 39.58, -64.05, -19.007] to (-92.16, 498.42, -3.54) mm, rotated rx -180 ry 0 rz 0 deg; joints [34.958, -44.203, 102.966, 39.584, -64.027, -19.026]
  Set speed (500.0 mm/s)
  MoveL 191 to (-92.16, 498.42, 5) mm, rotated rx -180 ry 0 rz 0 deg; joints [34.954, -44.631, 102.979, 39.71, -63.705, -19.319]
  MoveL 192 to (-92.16, 499.69, 5) mm, rotated rx -180 ry 0 rz 0 deg; joints [34.994, -44.599, 102.91, 39.763, -63.691, -19.363]
  Set speed (25.4 mm/s)
  MoveL 193 to (-92.16, 499.69, 1.83) mm, rotated rx -180 ry 0 rz 0 deg; joints [34.995, -44.44, 102.906, 39.716, -63.81, -19.253]
  MoveL 194 to (-92.16, 499.69, -7.72) mm, rotated rx 180 ry 0 rz 0 deg; joints [35, -43.961, 102.89, 39.577, -64.168, -18.927]
  MoveC 195 to (-91.98, 499.69, -8.16) mm, rotated rx -180 ry 0 rz 0 deg; joints [35.004, -43.945, 102.903, 39.572, -64.192, -18.908] to (-91.53, 499.69, -8.35) mm, rotated rx 180 ry 0 rz 0 deg; joints [35.014, -43.952, 102.937, 39.574, -64.216, -18.893]
  Set speed (50.8 mm/s)
  MoveL 196 to (-90.89, 499.69, -8.35) mm, rotated rx 180 ry 0 rz 0 deg; joints [35.028, -43.976, 102.986, 39.581, -64.24, -18.881]
  MoveC 197 to (-90.44, 499.51, -8.35) mm, rotated rx -180 ry 0 rz 0 deg; joints [35.032, -43.997, 103.031, 39.578, -64.259, -18.867] to (-90.26, 499.06, -8.35) mm, rotated rx -180 ry 0 rz 0 deg; joints [35.022, -44.015, 103.069, 39.561, -64.271, -18.848]
  MoveL 198 to (-90.26, 473.66, -8.35) mm, rotated rx -180 ry 0 rz 0 deg; joints [34.223, -44.644, 104.415, 38.507, -64.573, -17.997]
  MoveL 199 to (-141.06, 473.66, -8.35) mm, rotated rx -180 ry 0 rz 0 deg; joints [33.157, -42.723, 100.426, 38.016, -62.606, -18.942]
  MoveL 200 to (-141.06, 524.46, -8.35) mm, rotated rx -180 ry 0 rz 0 deg; joints [34.716, -41.429, 97.673, 40.152, -62.009, -20.726]
  MoveL 201 to (-90.26, 524.46, -8.35) mm, rotated rx -180 ry 0 rz 0 deg; joints [35.805, -43.365, 101.681, 40.612, -63.968, -19.723]
  MoveL 202 to (-90.26, 499.06, -8.35) mm, rotated rx -180 ry 0 rz 0 deg; joints [35.022, -44.015, 103.069, 39.561, -64.271, -18.848]
  MoveC 203 to (-90.44, 498.61, -8.35) mm, rotated rx -180 ry 0 rz 0 deg; joints [35.004, -44.02, 103.079, 39.541, -64.27, -18.836] to (-90.89, 498.42, -8.35) mm, rotated rx 180 ry 0 rz 0 deg; joints [34.988, -44.008, 103.055, 39.528, -64.255, -18.838]
  MoveL 204 to (-91.53, 498.42, -8.35) mm, rotated rx -180 ry 0 rz 0 deg; joints [34.974, -43.984, 103.006, 39.522, -64.231, -18.85]
  MoveC 205 to (-91.98, 498.42, -8.16) mm, rotated rx 180 ry 0 rz 0 deg; joints [34.965, -43.977, 102.972, 39.52, -64.207, -18.865] to (-92.16, 498.42, -7.72) mm, rotated rx -180 ry 0 rz 0 deg; joints [34.96, -43.993, 102.958, 39.524, -64.183, -18.883]
  Set speed (500.0 mm/s)
  MoveL 206 to (-92.16, 498.42, 6) mm, rotated rx 180 ry 0 rz 0 deg; joints [34.954, -44.681, 102.98, 39.725, -63.667, -19.354]
  MoveL 207 to (-219.16, 499.69, 6) mm, rotated rx 180 ry 0 rz 0 deg; joints [32.409, -39.564, 92.515, 38.877, -58.619, -21.95]
  Set speed (25.4 mm/s)
  MoveL 208 to (-219.16, 499.69, -3.54) mm, rotated rx -180 ry 0 rz 0 deg; joints [32.413, -39.126, 92.502, 38.72, -58.951, -21.641]
  MoveC 209 to (-218.98, 499.69, -3.99) mm, rotated rx -180 ry 0 rz 0 deg; joints [32.417, -39.113, 92.517, 38.713, -58.975, -21.622] to (-218.53, 499.69, -4.17) mm, rotated rx -180 ry 0 rz 0 deg; joints [32.426, -39.123, 92.556, 38.712, -59, -21.606]
  Set speed (50.8 mm/s)
  MoveL 210 to (-217.89, 499.69, -4.18) mm, rotated rx 180 ry 0 rz 0 deg; joints [32.438, -39.15, 92.611, 38.715, -59.027, -21.592]
  MoveC 211 to (-217.44, 499.51, -4.18) mm, rotated rx -180 ry 0 rz 0 deg; joints [32.441, -39.174, 92.66, 38.708, -59.048, -21.575] to (-217.26, 499.06, -4.18) mm, rotated rx 180 ry 0 rz 0 deg; joints [32.431, -39.194, 92.702, 38.689, -59.061, -21.554]
  MoveL 212 to (-217.26, 473.66, -4.18) mm, rotated rx -180 ry 0 rz 0 deg; joints [31.663, -39.848, 94.081, 37.59, -59.352, -20.618]
  MoveL 213 to (-268.06, 473.66, -4.18) mm, rotated rx -180 ry 0 rz 0 deg; joints [30.733, -37.649, 89.56, 37.447, -57.17, -21.76]
  MoveL 214 to (-268.06, 524.46, -4.17) mm, rotated rx -180 ry 0 rz 0 deg; joints [32.232, -36.283, 86.693, 39.705, -56.582, -23.755]
  MoveL 215 to (-217.26, 524.46, -4.17) mm, rotated rx -180 ry 0 rz 0 deg; joints [33.186, -38.515, 91.273, 39.791, -58.767, -22.518]
  MoveL 216 to (-217.26, 499.06, -4.18) mm, rotated rx 180 ry 0 rz 0 deg; joints [32.431, -39.194, 92.702, 38.689, -59.061, -21.554]
  MoveC 217 to (-217.44, 498.61, -4.18) mm, rotated rx 180 ry 0 rz 0 deg; joints [32.414, -39.198, 92.71, 38.669, -59.058, -21.542] to (-217.89, 498.42, -4.17) mm, rotated rx 180 ry 0 rz 0 deg; joints [32.4, -39.183, 92.681, 38.66, -59.042, -21.545]
  MoveL 218 to (-218.53, 498.42, -4.17) mm, rotated rx 180 ry 0 rz 0 deg; joints [32.387, -39.157, 92.626, 38.657, -59.015, -21.559]
  MoveC 219 to (-218.98, 498.42, -3.99) mm, rotated rx 180 ry 0 rz 0 deg; joints [32.379, -39.146, 92.587, 38.658, -58.989, -21.575] to (-219.16, 498.42, -3.54) mm, rotated rx 180 ry 0 rz 0 deg; joints [32.375, -39.159, 92.572, 38.665, -58.966, -21.593]
  Set speed (500.0 mm/s)
  MoveL 220 to (-219.16, 498.42, 5) mm, rotated rx -180 ry 0 rz 0 deg; joints [32.371, -39.552, 92.584, 38.805, -58.668, -21.87]
  MoveL 221 to (-219.16, 499.69, 5) mm, rotated rx -180 ry 0 rz 0 deg; joints [32.41, -39.518, 92.514, 38.86, -58.654, -21.917]
  Set speed (25.4 mm/s)
  MoveL 222 to (-219.16, 499.69, 1.82) mm, rotated rx 180 ry 0 rz 0 deg; joints [32.411, -39.373, 92.51, 38.808, -58.765, -21.814]
  MoveL 223 to (-219.16, 499.69, -7.72) mm, rotated rx -180 ry 0 rz 0 deg; joints [32.415, -38.933, 92.493, 38.653, -59.096, -21.507]
  MoveC 224 to (-218.98, 499.69, -8.16) mm, rotated rx 180 ry 0 rz 0 deg; joints [32.419, -38.92, 92.509, 38.646, -59.12, -21.489] to (-218.53, 499.69, -8.35) mm, rotated rx -180 ry 0 rz 0 deg; joints [32.427, -38.93, 92.547, 38.645, -59.145, -21.473]
  Set speed (50.8 mm/s)
  MoveL 225 to (-217.89, 499.69, -8.35) mm, rotated rx -180 ry 0 rz 0 deg; joints [32.439, -38.957, 92.603, 38.647, -59.172, -21.458]
  MoveC 226 to (-217.44, 499.51, -8.35) mm, rotated rx 180 ry 0 rz 0 deg; joints [32.442, -38.981, 92.652, 38.641, -59.193, -21.441] to (-217.26, 499.06, -8.35) mm, rotated rx -180 ry 0 rz 0 deg; joints [32.433, -39, 92.693, 38.622, -59.206, -21.421]
  MoveL 227 to (-217.26, 473.66, -8.35) mm, rotated rx 180 ry 0 rz 0 deg; joints [31.665, -39.652, 94.072, 37.525, -59.501, -20.487]
  MoveL 228 to (-268.06, 473.66, -8.35) mm, rotated rx -180 ry 0 rz 0 deg; joints [30.735, -37.46, 89.551, 37.379, -57.314, -21.631]
  MoveL 229 to (-268.06, 524.46, -8.35) mm, rotated rx -180 ry 0 rz 0 deg; joints [32.233, -36.098, 86.685, 39.633, -56.719, -23.621]
  MoveL 230 to (-217.26, 524.46, -8.35) mm, rotated rx -180 ry 0 rz 0 deg; joints [33.188, -38.324, 91.265, 39.722, -58.908, -22.382]
  MoveL 231 to (-217.26, 499.06, -8.35) mm, rotated rx -180 ry 0 rz 0 deg; joints [32.433, -39, 92.693, 38.622, -59.206, -21.421]
  MoveC 232 to (-217.44, 498.61, -8.35) mm, rotated rx 180 ry 0 rz 0 deg; joints [32.415, -39.004, 92.702, 38.602, -59.203, -21.408] to (-217.89, 498.42, -8.35) mm, rotated rx 180 ry 0 rz 0 deg; joints [32.401, -38.99, 92.673, 38.592, -59.187, -21.411]
  MoveL 233 to (-218.53, 498.42, -8.35) mm, rotated rx 180 ry 0 rz 0 deg; joints [32.389, -38.963, 92.617, 38.59, -59.16, -21.425]
  MoveC 234 to (-218.98, 498.42, -8.16) mm, rotated rx -180 ry 0 rz 0 deg; joints [32.381, -38.953, 92.579, 38.591, -59.135, -21.441] to (-219.16, 498.42, -7.72) mm, rotated rx 180 ry 0 rz 0 deg; joints [32.377, -38.966, 92.564, 38.598, -59.111, -21.46]
  Set speed (500.0 mm/s)
  MoveL 235 to (-219.16, 498.42, 6) mm, rotated rx -180 ry 0 rz 0 deg; joints [32.371, -39.598, 92.585, 38.822, -58.633, -21.902]
  MoveL 236 to (-346.16, 499.69, 6) mm, rotated rx 180 ry 0 rz 0 deg; joints [30.146, -33.701, 80.567, 38.973, -52.968, -25.2]
  Set speed (25.4 mm/s)
  MoveL 237 to (-346.16, 499.69, -3.54) mm, rotated rx 180 ry 0 rz 0 deg; joints [30.15, -33.297, 80.553, 38.793, -53.273, -24.896]
  MoveC 238 to (-345.98, 499.69, -3.99) mm, rotated rx -180 ry 0 rz 0 deg; joints [30.153, -33.287, 80.571, 38.784, -53.296, -24.876] to (-345.53, 499.69, -4.17) mm, rotated rx -180 ry 0 rz 0 deg; joints [30.161, -33.301, 80.616, 38.778, -53.324, -24.857]
  Set speed (50.8 mm/s)
  MoveL 239 to (-344.89, 499.69, -4.18) mm, rotated rx 180 ry 0 rz 0 deg; joints [30.172, -33.333, 80.681, 38.775, -53.354, -24.838]
  MoveC 240 to (-344.44, 499.51, -4.18) mm, rotated rx -180 ry 0 rz 0 deg; joints [30.174, -33.36, 80.738, 38.763, -53.378, -24.817] to (-344.26, 499.06, -4.17) mm, rotated rx 180 ry 0 rz 0 deg; joints [30.164, -33.382, 80.783, 38.741, -53.392, -24.792]
  MoveL 241 to (-344.26, 473.66, -4.18) mm, rotated rx 180 ry 0 rz 0 deg; joints [29.428, -34.086, 82.254, 37.559, -53.689, -23.72]
  MoveL 242 to (-395.06, 473.66, -4.17) mm, rotated rx -180 ry 0 rz 0 deg; joints [28.612, -31.494, 76.95, 37.9, -51.203, -25.255]
  MoveL 243 to (-395.06, 524.46, -4.17) mm, rotated rx 180 ry 0 rz 0 deg; joints [30.049, -29.985, 73.812, 40.391, -50.585, -27.602]
  MoveL 244 to (-344.26, 524.46, -4.17) mm, rotated rx 180 ry 0 rz 0 deg; joints [30.889, -32.648, 79.252, 39.935, -53.089, -25.9]
  MoveL 245 to (-344.26, 499.06, -4.17) mm, rotated rx 180 ry 0 rz 0 deg; joints [30.164, -33.382, 80.783, 38.741, -53.392, -24.792]
  MoveC 246 to (-344.44, 498.61, -4.18) mm, rotated rx -180 ry 0 rz 0 deg; joints [30.148, -33.386, 80.791, 38.721, -53.388, -24.778] to (-344.89, 498.42, -4.17) mm, rotated rx -180 ry 0 rz 0 deg; joints [30.135, -33.369, 80.756, 38.715, -53.369, -24.784]
  MoveL 247 to (-345.53, 498.42, -4.18) mm, rotated rx -180 ry 0 rz 0 deg; joints [30.124, -33.337, 80.691, 38.719, -53.339, -24.802]
  MoveC 248 to (-345.98, 498.42, -3.99) mm, rotated rx -180 ry 0 rz 0 deg; joints [30.117, -33.323, 80.646, 38.724, -53.311, -24.822] to (-346.16, 498.42, -3.54) mm, rotated rx -180 ry 0 rz 0 deg; joints [30.114, -33.333, 80.628, 38.734, -53.288, -24.841]
  Set speed (500.0 mm/s)
  MoveL 249 to (-346.16, 498.42, 5) mm, rotated rx 180 ry 0 rz 0 deg; joints [30.11, -33.695, 80.641, 38.894, -53.014, -25.113]
  MoveL 250 to (-346.16, 499.69, 5) mm, rotated rx 180 ry 0 rz 0 deg; joints [30.147, -33.659, 80.566, 38.954, -53, -25.168]
  Set speed (25.4 mm/s)
  MoveL 251 to (-346.16, 499.69, 1.82) mm, rotated rx 180 ry 0 rz 0 deg; joints [30.148, -33.525, 80.562, 38.894, -53.102, -25.066]
  MoveL 252 to (-346.16, 499.69, -7.72) mm, rotated rx -180 ry 0 rz 0 deg; joints [30.152, -33.118, 80.544, 38.716, -53.406, -24.765]
  MoveC 253 to (-345.98, 499.69, -8.16) mm, rotated rx 180 ry 0 rz 0 deg; joints [30.155, -33.108, 80.562, 38.707, -53.429, -24.745] to (-345.53, 499.69, -8.35) mm, rotated rx -180 ry 0 rz 0 deg; joints [30.163, -33.123, 80.607, 38.701, -53.457, -24.726]
  Set speed (50.8 mm/s)
  MoveL 254 to (-344.89, 499.69, -8.35) mm, rotated rx -180 ry 0 rz 0 deg; joints [30.173, -33.154, 80.672, 38.698, -53.487, -24.707]
  MoveC 255 to (-344.44, 499.51, -8.35) mm, rotated rx -180 ry 0 rz 0 deg; joints [30.175, -33.182, 80.729, 38.687, -53.511, -24.686] to (-344.26, 499.06, -8.35) mm, rotated rx -180 ry 0 rz 0 deg; joints [30.166, -33.204, 80.774, 38.665, -53.525, -24.661]
  MoveL 256 to (-344.26, 473.66, -8.35) mm, rotated rx -180 ry 0 rz 0 deg; joints [29.429, -33.906, 82.245, 37.484, -53.825, -23.591]
  MoveL 257 to (-395.06, 473.66, -8.35) mm, rotated rx -180 ry 0 rz 0 deg; joints [28.614, -31.319, 76.941, 37.821, -51.334, -25.126]
  MoveL 258 to (-395.06, 524.46, -8.35) mm, rotated rx -180 ry 0 rz 0 deg; joints [30.051, -29.813, 73.803, 40.306, -50.71, -27.467]
  MoveL 259 to (-344.26, 524.46, -8.35) mm, rotated rx -180 ry 0 rz 0 deg; joints [30.891, -32.471, 79.243, 39.856, -53.219, -25.767]
  MoveL 260 to (-344.26, 499.06, -8.35) mm, rotated rx -180 ry 0 rz 0 deg; joints [30.166, -33.204, 80.774, 38.665, -53.525, -24.661]
  MoveC 261 to (-344.44, 498.61, -8.35) mm, rotated rx -180 ry 0 rz 0 deg; joints [30.149, -33.207, 80.782, 38.645, -53.521, -24.647] to (-344.89, 498.42, -8.35) mm, rotated rx -180 ry 0 rz 0 deg; joints [30.137, -33.19, 80.747, 38.638, -53.502, -24.653]
  MoveL 262 to (-345.53, 498.42, -8.35) mm, rotated rx 180 ry 0 rz 0 deg; joints [30.126, -33.159, 80.682, 38.642, -53.472, -24.671]
  MoveC 263 to (-345.98, 498.42, -8.16) mm, rotated rx -180 ry 0 rz 0 deg; joints [30.118, -33.144, 80.637, 38.647, -53.444, -24.69] to (-346.16, 498.42, -7.72) mm, rotated rx 180 ry 0 rz 0 deg; joints [30.115, -33.154, 80.619, 38.657, -53.421, -24.71]
  Set speed (500.0 mm/s)
  MoveL 264 to (-346.16, 498.42, 6) mm, rotated rx -180 ry 0 rz 0 deg; joints [30.11, -33.738, 80.642, 38.913, -52.982, -25.145]
  MoveL 265 to (139.15, 499.69, 6) mm, rotated rx 180 ry 0 rz 0 deg; joints [40.731, -52.508, 119.071, 43.428, -71.621, -15.598]
  Set speed (25.4 mm/s)
  MoveL 266 to (139.15, 499.69, -3.54) mm, rotated rx -180 ry 0 rz 0 deg; joints [40.737, -51.942, 119.057, 43.309, -72.024, -15.2]
  MoveC 267 to (139.34, 499.69, -3.99) mm, rotated rx 180 ry 0 rz 0 deg; joints [40.742, -51.921, 119.068, 43.308, -72.049, -15.178] to (139.79, 499.69, -4.17) mm, rotated rx -180 ry 0 rz 0 deg; joints [40.755, -51.923, 119.096, 43.315, -72.071, -15.164]
  Set speed (50.8 mm/s)
  MoveL 268 to (140.42, 499.69, -4.18) mm, rotated rx 180 ry 0 rz 0 deg; joints [40.773, -51.942, 119.137, 43.329, -72.091, -15.154]
  MoveC 269 to (140.87, 499.51, -4.18) mm, rotated rx -180 ry 0 rz 0 deg; joints [40.779, -51.96, 119.175, 43.331, -72.107, -15.141] to (141.06, 499.06, -4.17) mm, rotated rx 180 ry 0 rz 0 deg; joints [40.77, -51.977, 119.211, 43.317, -72.119, -15.124]
  MoveL 270 to (141.06, 473.66, -4.18) mm, rotated rx -180 ry 0 rz 0 deg; joints [39.927, -52.602, 120.579, 42.301, -72.446, -14.347]
  MoveL 271 to (90.26, 473.66, -4.17) mm, rotated rx -180 ry 0 rz 0 deg; joints [38.541, -51.032, 117.284, 41.272, -70.8, -15.135]
  MoveL 272 to (90.26, 524.46, -4.17) mm, rotated rx 180 ry 0 rz 0 deg; joints [40.191, -49.767, 114.536, 43.307, -70.164, -16.73]
  MoveL 273 to (141.06, 524.46, -4.17) mm, rotated rx -180 ry 0 rz 0 deg; joints [41.592, -51.334, 117.809, 44.32, -71.795, -15.923]
  MoveL 274 to (141.06, 499.06, -4.17) mm, rotated rx 180 ry 0 rz 0 deg; joints [40.77, -51.977, 119.211, 43.317, -72.119, -15.124]
  MoveC 275 to (140.87, 498.61, -4.17) mm, rotated rx 180 ry 0 rz 0 deg; joints [40.75, -51.983, 119.224, 43.295, -72.119, -15.113] to (140.42, 498.42, -4.17) mm, rotated rx -180 ry 0 rz 0 deg; joints [40.731, -51.974, 119.206, 43.278, -72.107, -15.115]
  MoveL 276 to (139.79, 498.42, -4.17) mm, rotated rx 180 ry 0 rz 0 deg; joints [40.713, -51.955, 119.166, 43.265, -72.087, -15.124]
  MoveC 277 to (139.34, 498.42, -3.99) mm, rotated rx -180 ry 0 rz 0 deg; joints [40.701, -51.952, 119.137, 43.257, -72.065, -15.139] to (139.15, 498.42, -3.54) mm, rotated rx 180 ry 0 rz 0 deg; joints [40.695, -51.973, 119.127, 43.259, -72.04, -15.161]
  Set speed (500.0 mm/s)
  MoveL 278 to (139.15, 498.42, 5) mm, rotated rx -180 ry 0 rz 0 deg; joints [40.69, -52.481, 119.139, 43.365, -71.679, -15.516]
  MoveL 279 to (139.15, 499.69, 5) mm, rotated rx -180 ry 0 rz 0 deg; joints [40.732, -52.449, 119.07, 43.416, -71.663, -15.556]
  Set speed (25.4 mm/s)
  MoveL 280 to (139.15, 499.69, 1.82) mm, rotated rx -180 ry 0 rz 0 deg; joints [40.734, -52.26, 119.066, 43.376, -71.798, -15.423]
  MoveL 281 to (139.15, 499.69, -7.72) mm, rotated rx -180 ry 0 rz 0 deg; joints [40.739, -51.693, 119.049, 43.259, -72.2, -15.027]
  MoveC 282 to (139.34, 499.69, -8.16) mm, rotated rx -180 ry 0 rz 0 deg; joints [40.745, -51.672, 119.06, 43.257, -72.224, -15.006] to (139.79, 499.69, -8.35) mm, rotated rx -180 ry 0 rz 0 deg; joints [40.757, -51.674, 119.088, 43.264, -72.246, -14.991]
  Set speed (50.8 mm/s)
  MoveL 283 to (140.42, 499.69, -8.35) mm, rotated rx -180 ry 0 rz 0 deg; joints [40.775, -51.693, 119.128, 43.278, -72.266, -14.981]
  MoveC 284 to (140.87, 499.51, -8.35) mm, rotated rx -180 ry 0 rz 0 deg; joints [40.782, -51.711, 119.166, 43.28, -72.283, -14.969] to (141.06, 499.06, -8.35) mm, rotated rx -180 ry 0 rz 0 deg; joints [40.772, -51.728, 119.203, 43.266, -72.295, -14.952]
  MoveL 285 to (141.06, 473.66, -8.35) mm, rotated rx -180 ry 0 rz 0 deg; joints [39.93, -52.348, 120.57, 42.252, -72.628, -14.175]
  MoveL 286 to (90.26, 473.66, -8.35) mm, rotated rx -180 ry 0 rz 0 deg; joints [38.544, -50.789, 117.276, 41.221, -70.978, -14.972]
  MoveL 287 to (90.26, 524.46, -8.35) mm, rotated rx -180 ry 0 rz 0 deg; joints [40.194, -49.53, 114.527, 43.254, -70.33, -16.565]
  MoveL 288 to (141.06, 524.46, -8.35) mm, rotated rx -180 ry 0 rz 0 deg; joints [41.594, -51.089, 117.8, 44.268, -71.965, -15.749]
  MoveL 289 to (141.06, 499.06, -8.35) mm, rotated rx -180 ry 0 rz 0 deg; joints [40.772, -51.728, 119.203, 43.266, -72.295, -14.952]
  MoveC 290 to (140.87, 498.61, -8.35) mm, rotated rx -180 ry 0 rz 0 deg; joints [40.752, -51.733, 119.215, 43.245, -72.295, -14.941] to (140.42, 498.42, -8.35) mm, rotated rx -180 ry 0 rz 0 deg; joints [40.734, -51.724, 119.197, 43.228, -72.283, -14.942]
  MoveL 291 to (139.79, 498.42, -8.35) mm, rotated rx -180 ry 0 rz 0 deg; joints [40.716, -51.705, 119.157, 43.214, -72.263, -14.952]
  MoveC 292 to (139.34, 498.42, -8.16) mm, rotated rx 180 ry 0 rz 0 deg; joints [40.703, -51.703, 119.129, 43.207, -72.241, -14.967] to (139.15, 498.42, -7.72) mm, rotated rx 180 ry 0 rz 0 deg; joints [40.697, -51.724, 119.118, 43.208, -72.216, -14.988]
  Set speed (500.0 mm/s)
  MoveL 293 to (139.15, 498.42, 6) mm, rotated rx -180 ry 0 rz 0 deg; joints [40.689, -52.54, 119.14, 43.378, -71.636, -15.558]
  MoveL 294 to (266.15, 499.69, 6) mm, rotated rx -180 ry 0 rz 0 deg; joints [44.584, -56.199, 126.713, 46.486, -75.411, -13.729]
  Set speed (25.4 mm/s)
  MoveL 295 to (266.15, 499.69, -3.54) mm, rotated rx 180 ry 0 rz 0 deg; joints [44.59, -55.574, 126.699, 46.378, -75.834, -13.273]
  MoveC 296 to (266.34, 499.69, -3.99) mm, rotated rx -180 ry 0 rz 0 deg; joints [44.596, -55.549, 126.709, 46.378, -75.859, -13.249] to (266.79, 499.69, -4.17) mm, rotated rx -180 ry 0 rz 0 deg; joints [44.611, -55.549, 126.734, 46.389, -75.88, -13.233]
  Set speed (50.8 mm/s)
  MoveL 297 to (267.42, 499.69, -4.17) mm, rotated rx -180 ry 0 rz 0 deg; joints [44.632, -55.566, 126.77, 46.406, -75.898, -13.224]
  MoveC 298 to (267.87, 499.51, -4.17) mm, rotated rx -180 ry 0 rz 0 deg; joints [44.64, -55.583, 126.806, 46.411, -75.913, -13.212] to (268.06, 499.06, -4.18) mm, rotated rx -180 ry 0 rz 0 deg; joints [44.632, -55.599, 126.842, 46.399, -75.925, -13.195]
  MoveL 299 to (268.06, 473.66, -4.17) mm, rotated rx -180 ry 0 rz 0 deg; joints [43.778, -56.231, 128.252, 45.404, -76.273, -12.427]
  MoveL 300 to (217.26, 473.66, -4.17) mm, rotated rx -180 ry 0 rz 0 deg; joints [42.168, -54.829, 125.277, 44.07, -74.792, -13.189]
  MoveL 301 to (217.26, 524.46, -4.18) mm, rotated rx 180 ry 0 rz 0 deg; joints [43.847, -53.554, 122.462, 46.062, -74.117, -14.748]
  MoveL 302 to (268.06, 524.46, -4.17) mm, rotated rx -180 ry 0 rz 0 deg; joints [45.461, -54.949, 125.4, 47.376, -75.582, -13.983]
  MoveL 303 to (268.06, 499.06, -4.18) mm, rotated rx -180 ry 0 rz 0 deg; joints [44.632, -55.599, 126.842, 46.399, -75.925, -13.195]
  MoveC 304 to (267.87, 498.61, -4.17) mm, rotated rx -180 ry 0 rz 0 deg; joints [44.611, -55.606, 126.856, 46.376, -75.925, -13.184] to (267.42, 498.42, -4.17) mm, rotated rx -180 ry 0 rz 0 deg; joints [44.59, -55.598, 126.841, 46.357, -75.915, -13.185]
  MoveL 305 to (266.79, 498.42, -4.18) mm, rotated rx -180 ry 0 rz 0 deg; joints [44.569, -55.581, 126.805, 46.339, -75.897, -13.195]
  MoveC 306 to (266.34, 498.42, -3.99) mm, rotated rx 180 ry 0 rz 0 deg; joints [44.554, -55.581, 126.78, 46.329, -75.876, -13.21] to (266.15, 498.42, -3.54) mm, rotated rx 180 ry 0 rz 0 deg; joints [44.548, -55.606, 126.77, 46.329, -75.851, -13.234]
  Set speed (500.0 mm/s)
  MoveL 307 to (266.15, 498.42, 5) mm, rotated rx -180 ry 0 rz 0 deg; joints [44.542, -56.167, 126.783, 46.425, -75.472, -13.642]
  MoveL 308 to (266.15, 499.69, 5) mm, rotated rx -180 ry 0 rz 0 deg; joints [44.584, -56.134, 126.712, 46.474, -75.456, -13.681]
  Set speed (25.4 mm/s)
  MoveL 309 to (266.15, 499.69, 1.83) mm, rotated rx -180 ry 0 rz 0 deg; joints [44.586, -55.926, 126.708, 46.438, -75.596, -13.529]
  MoveL 310 to (266.15, 499.69, -7.71) mm, rotated rx -180 ry 0 rz 0 deg; joints [44.593, -55.299, 126.69, 46.333, -76.018, -13.075]
  MoveC 311 to (266.34, 499.69, -8.16) mm, rotated rx 180 ry 0 rz 0 deg; joints [44.599, -55.274, 126.7, 46.333, -76.043, -13.051] to (266.79, 499.69, -8.35) mm, rotated rx -180 ry 0 rz 0 deg; joints [44.614, -55.274, 126.725, 46.343, -76.064, -13.036]
  Set speed (50.8 mm/s)
  MoveL 312 to (267.42, 499.69, -8.35) mm, rotated rx -180 ry 0 rz 0 deg; joints [44.635, -55.291, 126.761, 46.36, -76.082, -13.026]
  MoveC 313 to (267.87, 499.51, -8.35) mm, rotated rx 180 ry 0 rz 0 deg; joints [44.643, -55.308, 126.797, 46.366, -76.098, -13.013] to (268.06, 499.06, -8.35) mm, rotated rx 180 ry 0 rz 0 deg; joints [44.634, -55.324, 126.833, 46.353, -76.109, -12.997]
  MoveL 314 to (268.06, 473.66, -8.35) mm, rotated rx -180 ry 0 rz 0 deg; joints [43.781, -55.95, 128.242, 45.36, -76.464, -12.228]
  MoveL 315 to (217.26, 473.66, -8.35) mm, rotated rx -180 ry 0 rz 0 deg; joints [42.171, -54.559, 125.268, 44.024, -74.98, -13.002]
  MoveL 316 to (217.26, 524.46, -8.35) mm, rotated rx -180 ry 0 rz 0 deg; joints [43.849, -53.294, 122.454, 46.013, -74.292, -14.561]
  MoveL 317 to (268.06, 524.46, -8.35) mm, rotated rx -180 ry 0 rz 0 deg; joints [45.463, -54.679, 125.391, 47.329, -75.759, -13.786]
  MoveL 318 to (268.06, 499.06, -8.35) mm, rotated rx 180 ry 0 rz 0 deg; joints [44.634, -55.324, 126.833, 46.353, -76.109, -12.997]
  MoveC 319 to (267.87, 498.61, -8.35) mm, rotated rx -180 ry 0 rz 0 deg; joints [44.613, -55.33, 126.847, 46.331, -76.11, -12.986] to (267.42, 498.42, -8.35) mm, rotated rx -180 ry 0 rz 0 deg; joints [44.592, -55.323, 126.832, 46.311, -76.1, -12.987]
  MoveL 320 to (266.79, 498.42, -8.35) mm, rotated rx -180 ry 0 rz 0 deg; joints [44.572, -55.306, 126.796, 46.294, -76.082, -12.997]
  MoveC 321 to (266.34, 498.42, -8.16) mm, rotated rx -180 ry 0 rz 0 deg; joints [44.557, -55.306, 126.771, 46.284, -76.061, -13.012] to (266.15, 498.42, -7.72) mm, rotated rx -180 ry 0 rz 0 deg; joints [44.551, -55.331, 126.761, 46.283, -76.036, -13.036]
  Set speed (500.0 mm/s)
  MoveL 322 to (266.15, 498.42, 6) mm, rotated rx 180 ry 0 rz 0 deg; joints [44.542, -56.232, 126.784, 46.436, -75.428, -13.69]
  MoveL 323 to (393.15, 499.69, 6) mm, rotated rx -180 ry 0 rz 0 deg; joints [49.044, -59.487, 133.553, 50.335, -78.783, -11.929]
  Set speed (25.4 mm/s)
  MoveL 324 to (393.15, 499.69, -3.54) mm, rotated rx 180 ry 0 rz 0 deg; joints [49.051, -58.794, 133.538, 50.24, -79.218, -11.399]
  MoveC 325 to (393.34, 499.69, -3.99) mm, rotated rx 180 ry 0 rz 0 deg; joints [49.058, -58.765, 133.547, 50.242, -79.243, -11.371] to (393.79, 499.69, -4.17) mm, rotated rx -180 ry 0 rz 0 deg; joints [49.075, -58.762, 133.569, 50.255, -79.262, -11.354]
  Set speed (50.8 mm/s)
  MoveL 326 to (394.42, 499.69, -4.17) mm, rotated rx 180 ry 0 rz 0 deg; joints [49.099, -58.777, 133.601, 50.277, -79.278, -11.345]
  MoveC 327 to (394.87, 499.51, -4.17) mm, rotated rx -180 ry 0 rz 0 deg; joints [49.11, -58.793, 133.635, 50.285, -79.292, -11.333] to (395.06, 499.06, -4.17) mm, rotated rx -180 ry 0 rz 0 deg; joints [49.103, -58.809, 133.671, 50.274, -79.303, -11.316]
  MoveL 328 to (395.06, 473.66, -4.17) mm, rotated rx -180 ry 0 rz 0 deg; joints [48.256, -59.452, 135.139, 49.313, -79.671, -10.534]
  MoveL 329 to (344.26, 473.66, -4.17) mm, rotated rx 180 ry 0 rz 0 deg; joints [46.383, -58.213, 132.478, 47.648, -78.365, -11.29]
  MoveL 330 to (344.26, 524.46, -4.18) mm, rotated rx -180 ry 0 rz 0 deg; joints [48.061, -56.918, 129.562, 49.582, -77.652, -12.856]
  MoveL 331 to (395.06, 524.46, -4.18) mm, rotated rx 180 ry 0 rz 0 deg; joints [49.921, -58.148, 132.174, 51.214, -78.944, -12.117]
  MoveL 332 to (395.06, 499.06, -4.17) mm, rotated rx -180 ry 0 rz 0 deg; joints [49.103, -58.809, 133.671, 50.274, -79.303, -11.316]
  MoveC 333 to (394.87, 498.61, -4.17) mm, rotated rx -180 ry 0 rz 0 deg; joints [49.081, -58.816, 133.687, 50.251, -79.305, -11.305] to (394.42, 498.42, -4.18) mm, rotated rx 180 ry 0 rz 0 deg; joints [49.058, -58.81, 133.676, 50.229, -79.296, -11.305]
  MoveL 334 to (393.79, 498.42, -4.17) mm, rotated rx -180 ry 0 rz 0 deg; joints [49.034, -58.795, 133.643, 50.208, -79.28, -11.315]
  MoveC 335 to (393.34, 498.42, -3.99) mm, rotated rx -180 ry 0 rz 0 deg; joints [49.017, -58.798, 133.621, 50.194, -79.261, -11.332] to (393.15, 498.42, -3.54) mm, rotated rx -180 ry 0 rz 0 deg; joints [49.009, -58.826, 133.612, 50.192, -79.236, -11.359]
  Set speed (500.0 mm/s)
  MoveL 336 to (393.15, 498.42, 5) mm, rotated rx -180 ry 0 rz 0 deg; joints [49.003, -59.448, 133.626, 50.277, -78.846, -11.834]
  MoveL 337 to (393.15, 499.69, 5) mm, rotated rx -180 ry 0 rz 0 deg; joints [49.045, -59.414, 133.552, 50.324, -78.828, -11.873]
  Set speed (25.4 mm/s)
  MoveL 338 to (393.15, 499.69, 1.82) mm, rotated rx -180 ry 0 rz 0 deg; joints [49.047, -59.184, 133.548, 50.293, -78.973, -11.696]
  MoveL 339 to (393.15, 499.69, -7.72) mm, rotated rx 180 ry 0 rz 0 deg; joints [49.054, -58.489, 133.529, 50.2, -79.407, -11.168]
  MoveC 340 to (393.34, 499.69, -8.16) mm, rotated rx 180 ry 0 rz 0 deg; joints [49.061, -58.461, 133.537, 50.202, -79.432, -11.141] to (393.79, 499.69, -8.35) mm, rotated rx -180 ry 0 rz 0 deg; joints [49.078, -58.458, 133.56, 50.216, -79.452, -11.124]
  Set speed (50.8 mm/s)
  MoveL 341 to (394.42, 499.69, -8.35) mm, rotated rx 180 ry 0 rz 0 deg; joints [49.102, -58.472, 133.592, 50.237, -79.467, -11.114]
  MoveC 342 to (394.87, 499.51, -8.35) mm, rotated rx -180 ry 0 rz 0 deg; joints [49.113, -58.488, 133.625, 50.245, -79.481, -11.102] to (395.06, 499.06, -8.35) mm, rotated rx -180 ry 0 rz 0 deg; joints [49.106, -58.503, 133.661, 50.235, -79.493, -11.085]
  MoveL 343 to (395.06, 473.66, -8.35) mm, rotated rx -180 ry 0 rz 0 deg; joints [48.259, -59.139, 135.129, 49.274, -79.869, -10.301]
  MoveL 344 to (344.26, 473.66, -8.35) mm, rotated rx -180 ry 0 rz 0 deg; joints [46.386, -57.913, 132.469, 47.607, -78.562, -11.072]
  MoveL 345 to (344.26, 524.46, -8.35) mm, rotated rx 180 ry 0 rz 0 deg; joints [48.064, -56.632, 129.553, 49.539, -77.832, -12.641]
  MoveL 346 to (395.06, 524.46, -8.35) mm, rotated rx -180 ry 0 rz 0 deg; joints [49.924, -57.85, 132.164, 51.174, -79.125, -11.888]
  MoveL 347 to (395.06, 499.06, -8.35) mm, rotated rx 180 ry 0 rz 0 deg; joints [49.106, -58.503, 133.661, 50.235, -79.493, -11.085]
  MoveC 348 to (394.87, 498.61, -8.35) mm, rotated rx -180 ry 0 rz 0 deg; joints [49.084, -58.51, 133.678, 50.212, -79.494, -11.074] to (394.42, 498.42, -8.35) mm, rotated rx 180 ry 0 rz 0 deg; joints [49.061, -58.505, 133.666, 50.19, -79.486, -11.075]
  MoveL 349 to (393.79, 498.42, -8.35) mm, rotated rx -180 ry 0 rz 0 deg; joints [49.037, -58.49, 133.634, 50.168, -79.47, -11.084]
  MoveC 350 to (393.34, 498.42, -8.16) mm, rotated rx -180 ry 0 rz 0 deg; joints [49.02, -58.493, 133.611, 50.155, -79.451, -11.101] to (393.15, 498.42, -7.72) mm, rotated rx 180 ry 0 rz 0 deg; joints [49.012, -58.521, 133.603, 50.153, -79.426, -11.129]
  Set speed (500.0 mm/s)
  MoveL 351 to (393.15, 498.42, 6) mm, rotated rx -180 ry 0 rz 0 deg; joints [49.002, -59.52, 133.627, 50.287, -78.8, -11.89]
  MoveL 352 to (393.15, 313.35, 6) mm, rotated rx -180 ry 0 rz 0 deg; joints [42.117, -63.936, 143.634, 42.683, -81.513, -6.692]
  Set speed (25.4 mm/s)
  MoveL 353 to (393.15, 313.36, -3.54) mm, rotated rx 180 ry 0 rz 0 deg; joints [42.125, -63.104, 143.616, 42.611, -82.113, -6.136]
  MoveC 354 to (393.34, 313.36, -3.99) mm, rotated rx -180 ry 0 rz 0 deg; joints [42.132, -63.069, 143.625, 42.615, -82.146, -6.107] to (393.79, 313.36, -4.17) mm, rotated rx 180 ry 0 rz 0 deg; joints [42.149, -63.064, 143.649, 42.629, -82.17, -6.089]
  Set speed (50.8 mm/s)
  MoveL 355 to (394.42, 313.35, -4.17) mm, rotated rx 180 ry 0 rz 0 deg; joints [42.173, -63.079, 143.684, 42.651, -82.187, -6.078]
  MoveC 356 to (394.87, 313.17, -4.17) mm, rotated rx -180 ry 0 rz 0 deg; joints [42.183, -63.094, 143.718, 42.659, -82.202, -6.066] to (395.06, 312.72, -4.18) mm, rotated rx -180 ry 0 rz 0 deg; joints [42.171, -63.107, 143.751, 42.645, -82.214, -6.052]
  MoveL 357 to (395.06, 287.32, -4.17) mm, rotated rx -180 ry 0 rz 0 deg; joints [41.086, -63.615, 144.996, 41.491, -82.649, -5.426]
  MoveL 358 to (344.26, 287.32, -4.17) mm, rotated rx -180 ry 0 rz 0 deg; joints [39.234, -62.345, 142.118, 39.78, -81.231, -6.252]
  MoveL 359 to (344.26, 338.12, -4.18) mm, rotated rx 180 ry 0 rz 0 deg; joints [41.35, -61.317, 139.659, 42.058, -80.413, -7.508]
  MoveL 360 to (395.06, 338.12, -4.17) mm, rotated rx -180 ry 0 rz 0 deg; joints [43.22, -62.58, 142.473, 43.77, -81.789, -6.702]
  MoveL 361 to (395.06, 312.72, -4.18) mm, rotated rx -180 ry 0 rz 0 deg; joints [42.171, -63.107, 143.751, 42.645, -82.214, -6.052]
  MoveC 362 to (394.87, 312.27, -4.18) mm, rotated rx 180 ry 0 rz 0 deg; joints [42.145, -63.112, 143.763, 42.619, -82.217, -6.044] to (394.42, 312.08, -4.17) mm, rotated rx 180 ry 0 rz 0 deg; joints [42.12, -63.105, 143.747, 42.594, -82.208, -6.046]
  MoveL 363 to (393.79, 312.08, -4.17) mm, rotated rx -180 ry 0 rz 0 deg; joints [42.096, -63.09, 143.712, 42.572, -82.191, -6.057]
  MoveC 364 to (393.34, 312.08, -3.99) mm, rotated rx 180 ry 0 rz 0 deg; joints [42.079, -63.095, 143.688, 42.558, -82.168, -6.075] to (393.15, 312.09, -3.54) mm, rotated rx 180 ry 0 rz 0 deg; joints [42.071, -63.13, 143.679, 42.554, -82.134, -6.104]
  Set speed (500.0 mm/s)
  MoveL 365 to (393.15, 312.08, 5) mm, rotated rx -180 ry 0 rz 0 deg; joints [42.065, -63.876, 143.695, 42.618, -81.596, -6.602]
  MoveL 366 to (393.15, 313.36, 5) mm, rotated rx -180 ry 0 rz 0 deg; joints [42.118, -63.849, 143.632, 42.675, -81.576, -6.634]
  Set speed (25.4 mm/s)
  MoveL 367 to (393.15, 313.36, 1.82) mm, rotated rx 180 ry 0 rz 0 deg; joints [42.121, -63.572, 143.627, 42.651, -81.776, -6.448]
  MoveL 368 to (393.15, 313.36, -7.72) mm, rotated rx -180 ry 0 rz 0 deg; joints [42.128, -62.738, 143.605, 42.582, -82.374, -5.894]
  MoveC 369 to (393.34, 313.36, -8.16) mm, rotated rx -180 ry 0 rz 0 deg; joints [42.135, -62.703, 143.614, 42.585, -82.407, -5.865] to (393.79, 313.36, -8.35) mm, rotated rx -180 ry 0 rz 0 deg; joints [42.153, -62.698, 143.638, 42.6, -82.431, -5.847]
  Set speed (50.8 mm/s)
  MoveL 370 to (394.42, 313.35, -8.35) mm, rotated rx -180 ry 0 rz 0 deg; joints [42.177, -62.713, 143.673, 42.622, -82.448, -5.836]
  MoveC 371 to (394.87, 313.17, -8.35) mm, rotated rx 180 ry 0 rz 0 deg; joints [42.186, -62.727, 143.707, 42.63, -82.463, -5.824] to (395.06, 312.72, -8.35) mm, rotated rx -180 ry 0 rz 0 deg; joints [42.174, -62.741, 143.739, 42.616, -82.476, -5.81]
  MoveL 372 to (395.06, 287.32, -8.35) mm, rotated rx 180 ry 0 rz 0 deg; joints [41.089, -63.239, 144.985, 41.464, -82.922, -5.183]
  MoveL 373 to (344.26, 287.32, -8.35) mm, rotated rx -180 ry 0 rz 0 deg; joints [39.237, -61.99, 142.107, 39.749, -81.495, -6.03]
  MoveL 374 to (344.26, 338.12, -8.35) mm, rotated rx -180 ry 0 rz 0 deg; joints [41.353, -60.979, 139.649, 42.024, -80.657, -7.286]
  MoveL 375 to (395.06, 338.12, -8.35) mm, rotated rx 180 ry 0 rz 0 deg; joints [43.223, -62.223, 142.462, 43.739, -82.039, -6.46]
  MoveL 376 to (395.06, 312.72, -8.35) mm, rotated rx -180 ry 0 rz 0 deg; joints [42.174, -62.741, 143.739, 42.616, -82.476, -5.81]
  MoveC 377 to (394.87, 312.27, -8.35) mm, rotated rx -180 ry 0 rz 0 deg; joints [42.148, -62.745, 143.751, 42.59, -82.479, -5.801] to (394.42, 312.09, -8.35) mm, rotated rx -180 ry 0 rz 0 deg; joints [42.123, -62.738, 143.736, 42.565, -82.47, -5.804]
  MoveL 378 to (393.79, 312.09, -8.35) mm, rotated rx 180 ry 0 rz 0 deg; joints [42.099, -62.723, 143.701, 42.543, -82.453, -5.815]
  MoveC 379 to (393.34, 312.08, -8.16) mm, rotated rx -180 ry 0 rz 0 deg; joints [42.082, -62.729, 143.677, 42.528, -82.429, -5.833] to (393.15, 312.09, -7.72) mm, rotated rx -180 ry 0 rz 0 deg; joints [42.075, -62.764, 143.668, 42.525, -82.396, -5.862]
  Set speed (500.0 mm/s)
  MoveL 380 to (393.15, 312.09, 6) mm, rotated rx -180 ry 0 rz 0 deg; joints [42.064, -63.963, 143.697, 42.626, -81.533, -6.661]
  MoveL 381 to (266.15, 313.36, 6) mm, rotated rx -180 ry 0 rz 0 deg; joints [37.718, -60.528, 136.303, 38.717, -77.931, -8.57]
  Set speed (25.4 mm/s)
  MoveL 382 to (266.15, 313.35, -3.54) mm, rotated rx -180 ry 0 rz 0 deg; joints [37.725, -59.802, 136.287, 38.631, -78.487, -8.118]
  MoveC 383 to (266.34, 313.35, -3.99) mm, rotated rx 180 ry 0 rz 0 deg; joints [37.731, -59.773, 136.297, 38.632, -78.518, -8.094] to (266.79, 313.36, -4.17) mm, rotated rx 180 ry 0 rz 0 deg; joints [37.745, -59.771, 136.324, 38.643, -78.543, -8.079]
  Set speed (50.8 mm/s)
  MoveL 384 to (267.42, 313.36, -4.18) mm, rotated rx -180 ry 0 rz 0 deg; joints [37.765, -59.789, 136.362, 38.661, -78.562, -8.069]
  MoveC 385 to (267.87, 313.17, -4.18) mm, rotated rx -180 ry 0 rz 0 deg; joints [37.772, -59.805, 136.398, 38.665, -78.578, -8.058] to (268.06, 312.72, -4.17) mm, rotated rx 180 ry 0 rz 0 deg; joints [37.76, -59.819, 136.43, 38.65, -78.591, -8.044]
  MoveL 386 to (268.06, 287.32, -4.18) mm, rotated rx 180 ry 0 rz 0 deg; joints [36.707, -60.318, 137.599, 37.506, -78.971, -7.432]
  MoveL 387 to (217.26, 287.32, -4.18) mm, rotated rx -180 ry 0 rz 0 deg; joints [35.173, -58.887, 134.454, 36.169, -77.384, -8.187]
  MoveL 388 to (217.26, 338.12, -4.17) mm, rotated rx -180 ry 0 rz 0 deg; joints [37.217, -57.878, 132.134, 38.424, -76.663, -9.437]
  MoveL 389 to (268.06, 338.12, -4.18) mm, rotated rx 180 ry 0 rz 0 deg; joints [38.783, -59.301, 135.227, 39.772, -78.213, -8.678]
  MoveL 390 to (268.06, 312.72, -4.18) mm, rotated rx -180 ry 0 rz 0 deg; joints [37.76, -59.819, 136.43, 38.65, -78.591, -8.044]
  MoveC 391 to (267.87, 312.27, -4.18) mm, rotated rx 180 ry 0 rz 0 deg; joints [37.735, -59.823, 136.44, 38.625, -78.592, -8.036] to (267.42, 312.09, -4.18) mm, rotated rx 180 ry 0 rz 0 deg; joints [37.714, -59.814, 136.421, 38.604, -78.581, -8.038]
  MoveL 392 to (266.79, 312.09, -4.18) mm, rotated rx -180 ry 0 rz 0 deg; joints [37.693, -59.796, 136.383, 38.587, -78.562, -8.048]
  MoveC 393 to (266.34, 312.08, -3.99) mm, rotated rx -180 ry 0 rz 0 deg; joints [37.679, -59.798, 136.356, 38.576, -78.537, -8.063] to (266.15, 312.09, -3.54) mm, rotated rx 180 ry 0 rz 0 deg; joints [37.673, -59.828, 136.346, 38.575, -78.505, -8.087]
  Set speed (500.0 mm/s)
  MoveL 394 to (266.15, 312.08, 5) mm, rotated rx 180 ry 0 rz 0 deg; joints [37.667, -60.478, 136.361, 38.651, -78.008, -8.491]
  MoveL 395 to (266.15, 313.36, 5) mm, rotated rx -180 ry 0 rz 0 deg; joints [37.719, -60.452, 136.302, 38.708, -77.99, -8.523]
  Set speed (25.4 mm/s)
  MoveL 396 to (266.15, 313.36, 1.83) mm, rotated rx -180 ry 0 rz 0 deg; joints [37.721, -60.211, 136.297, 38.679, -78.175, -8.372]
  MoveL 397 to (266.15, 313.35, -7.71) mm, rotated rx 180 ry 0 rz 0 deg; joints [37.728, -59.483, 136.277, 38.595, -78.728, -7.922]
  MoveC 398 to (266.34, 313.36, -8.16) mm, rotated rx -180 ry 0 rz 0 deg; joints [37.734, -59.454, 136.287, 38.597, -78.76, -7.898] to (266.79, 313.35, -8.35) mm, rotated rx -180 ry 0 rz 0 deg; joints [37.748, -59.452, 136.313, 38.607, -78.784, -7.883]
  Set speed (50.8 mm/s)
  MoveL 399 to (267.42, 313.36, -8.35) mm, rotated rx 180 ry 0 rz 0 deg; joints [37.768, -59.469, 136.352, 38.625, -78.804, -7.873]
  MoveC 400 to (267.87, 313.17, -8.35) mm, rotated rx -180 ry 0 rz 0 deg; joints [37.775, -59.485, 136.387, 38.629, -78.82, -7.861] to (268.06, 312.72, -8.35) mm, rotated rx 180 ry 0 rz 0 deg; joints [37.762, -59.499, 136.42, 38.614, -78.833, -7.847]
  MoveL 401 to (268.06, 287.32, -8.35) mm, rotated rx -180 ry 0 rz 0 deg; joints [36.71, -59.991, 137.588, 37.471, -79.222, -7.237]
  MoveL 402 to (217.26, 287.32, -8.35) mm, rotated rx 180 ry 0 rz 0 deg; joints [35.175, -58.577, 134.444, 36.133, -77.626, -8.007]
  MoveL 403 to (217.26, 338.12, -8.35) mm, rotated rx -180 ry 0 rz 0 deg; joints [37.22, -57.579, 132.124, 38.384, -76.89, -9.254]
  MoveL 404 to (268.06, 338.12, -8.35) mm, rotated rx -180 ry 0 rz 0 deg; joints [38.786, -58.988, 135.217, 39.735, -78.447, -8.481]
  MoveL 405 to (268.06, 312.72, -8.35) mm, rotated rx 180 ry 0 rz 0 deg; joints [37.762, -59.499, 136.42, 38.614, -78.833, -7.847]
  MoveC 406 to (267.87, 312.27, -8.35) mm, rotated rx -180 ry 0 rz 0 deg; joints [37.738, -59.503, 136.429, 38.589, -78.834, -7.839] to (267.42, 312.09, -8.35) mm, rotated rx -180 ry 0 rz 0 deg; joints [37.716, -59.494, 136.411, 38.569, -78.823, -7.842]
  MoveL 407 to (266.79, 312.08, -8.35) mm, rotated rx -180 ry 0 rz 0 deg; joints [37.696, -59.477, 136.372, 38.551, -78.804, -7.851]
  MoveC 408 to (266.34, 312.09, -8.16) mm, rotated rx -180 ry 0 rz 0 deg; joints [37.682, -59.479, 136.346, 38.54, -78.779, -7.867] to (266.15, 312.08, -7.72) mm, rotated rx -180 ry 0 rz 0 deg; joints [37.676, -59.508, 136.336, 38.539, -78.748, -7.891]
  Set speed (500.0 mm/s)
  MoveL 409 to (266.15, 312.09, 6) mm, rotated rx 180 ry 0 rz 0 deg; joints [37.667, -60.554, 136.362, 38.66, -77.949, -8.539]
  MoveL 410 to (139.15, 313.35, 6) mm, rotated rx -180 ry 0 rz 0 deg; joints [34.047, -56.745, 128.293, 35.625, -73.941, -10.353]
  Set speed (25.4 mm/s)
  MoveL 411 to (139.15, 313.35, -3.54) mm, rotated rx -180 ry 0 rz 0 deg; joints [34.053, -56.105, 128.278, 35.528, -74.45, -9.977]
  MoveC 412 to (139.34, 313.35, -3.99) mm, rotated rx -180 ry 0 rz 0 deg; joints [34.058, -56.081, 128.289, 35.528, -74.48, -9.956] to (139.79, 313.35, -4.17) mm, rotated rx 180 ry 0 rz 0 deg; joints [34.07, -56.082, 128.318, 35.536, -74.505, -9.943]
  Set speed (50.8 mm/s)
  MoveL 413 to (140.42, 313.35, -4.18) mm, rotated rx -180 ry 0 rz 0 deg; joints [34.087, -56.101, 128.36, 35.549, -74.526, -9.933]
  MoveC 414 to (140.87, 313.17, -4.17) mm, rotated rx 180 ry 0 rz 0 deg; joints [34.092, -56.119, 128.398, 35.551, -74.543, -9.922] to (141.06, 312.72, -4.17) mm, rotated rx -180 ry 0 rz 0 deg; joints [34.079, -56.133, 128.43, 35.535, -74.555, -9.908]
  MoveL 415 to (141.06, 287.32, -4.17) mm, rotated rx -180 ry 0 rz 0 deg; joints [33.072, -56.623, 129.539, 34.409, -74.891, -9.285]
  MoveL 416 to (90.26, 287.32, -4.18) mm, rotated rx -180 ry 0 rz 0 deg; joints [31.791, -55.036, 126.129, 33.388, -73.156, -10.001]
  MoveL 417 to (90.26, 338.12, -4.18) mm, rotated rx 180 ry 0 rz 0 deg; joints [33.743, -54.043, 123.91, 35.609, -72.515, -11.29]
  MoveL 418 to (141.06, 338.12, -4.17) mm, rotated rx -180 ry 0 rz 0 deg; joints [35.062, -55.625, 127.285, 36.644, -74.22, -10.553]
  MoveL 419 to (141.06, 312.72, -4.17) mm, rotated rx -180 ry 0 rz 0 deg; joints [34.079, -56.133, 128.43, 35.535, -74.555, -9.908]
  MoveC 420 to (140.87, 312.27, -4.17) mm, rotated rx -180 ry 0 rz 0 deg; joints [34.056, -56.136, 128.438, 35.511, -74.555, -9.9] to (140.42, 312.09, -4.18) mm, rotated rx -180 ry 0 rz 0 deg; joints [34.037, -56.126, 128.416, 35.493, -74.543, -9.902]
  MoveL 421 to (139.79, 312.08, -4.18) mm, rotated rx 180 ry 0 rz 0 deg; joints [34.02, -56.107, 128.375, 35.48, -74.522, -9.911]
  MoveC 422 to (139.34, 312.08, -3.99) mm, rotated rx 180 ry 0 rz 0 deg; joints [34.008, -56.105, 128.345, 35.472, -74.497, -9.925] to (139.15, 312.08, -3.54) mm, rotated rx -180 ry 0 rz 0 deg; joints [34.003, -56.13, 128.334, 35.472, -74.467, -9.945]
  Set speed (500.0 mm/s)
  MoveL 423 to (139.15, 312.08, 5) mm, rotated rx -180 ry 0 rz 0 deg; joints [33.998, -56.704, 128.348, 35.559, -74.01, -10.281]
  MoveL 424 to (139.15, 313.35, 5) mm, rotated rx -180 ry 0 rz 0 deg; joints [34.048, -56.678, 128.292, 35.615, -73.994, -10.313]
  Set speed (25.4 mm/s)
  MoveL 425 to (139.15, 313.36, 1.82) mm, rotated rx -180 ry 0 rz 0 deg; joints [34.05, -56.465, 128.287, 35.582, -74.164, -10.188]
  MoveL 426 to (139.15, 313.36, -7.71) mm, rotated rx -180 ry 0 rz 0 deg; joints [34.055, -55.824, 128.268, 35.487, -74.672, -9.813]
  MoveC 427 to (139.34, 313.35, -8.16) mm, rotated rx 180 ry 0 rz 0 deg; joints [34.061, -55.799, 128.28, 35.487, -74.702, -9.793] to (139.79, 313.35, -8.35) mm, rotated rx 180 ry 0 rz 0 deg; joints [34.073, -55.8, 128.309, 35.495, -74.727, -9.779]
  Set speed (50.8 mm/s)
  MoveL 428 to (140.42, 313.36, -8.35) mm, rotated rx -180 ry 0 rz 0 deg; joints [34.089, -55.819, 128.35, 35.508, -74.748, -9.77]
  MoveC 429 to (140.87, 313.17, -8.35) mm, rotated rx -180 ry 0 rz 0 deg; joints [34.094, -55.837, 128.388, 35.51, -74.765, -9.759] to (141.06, 312.72, -8.35) mm, rotated rx 180 ry 0 rz 0 deg; joints [34.081, -55.851, 128.42, 35.494, -74.778, -9.745]
  MoveL 430 to (141.06, 287.32, -8.35) mm, rotated rx -180 ry 0 rz 0 deg; joints [33.074, -56.337, 129.53, 34.37, -75.12, -9.123]
  MoveL 431 to (90.26, 287.32, -8.35) mm, rotated rx -180 ry 0 rz 0 deg; joints [31.794, -54.763, 126.119, 33.347, -73.377, -9.85]
  MoveL 432 to (90.26, 338.12, -8.35) mm, rotated rx 180 ry 0 rz 0 deg; joints [33.746, -53.778, 123.901, 35.565, -72.724, -11.135]
  MoveL 433 to (141.06, 338.12, -8.35) mm, rotated rx -180 ry 0 rz 0 deg; joints [35.065, -55.347, 127.275, 36.601, -74.436, -10.388]
  MoveL 434 to (141.06, 312.72, -8.35) mm, rotated rx 180 ry 0 rz 0 deg; joints [34.081, -55.851, 128.42, 35.494, -74.778, -9.745]
  MoveC 435 to (140.87, 312.27, -8.35) mm, rotated rx -180 ry 0 rz 0 deg; joints [34.059, -55.854, 128.428, 35.47, -74.778, -9.737] to (140.42, 312.09, -8.35) mm, rotated rx -180 ry 0 rz 0 deg; joints [34.04, -55.844, 128.407, 35.452, -74.765, -9.738]
  MoveL 436 to (139.79, 312.08, -8.35) mm, rotated rx 180 ry 0 rz 0 deg; joints [34.023, -55.825, 128.365, 35.439, -74.744, -9.748]
  MoveC 437 to (139.34, 312.08, -8.16) mm, rotated rx 180 ry 0 rz 0 deg; joints [34.011, -55.824, 128.336, 35.431, -74.719, -9.761] to (139.15, 312.08, -7.72) mm, rotated rx 180 ry 0 rz 0 deg; joints [34.006, -55.849, 128.325, 35.431, -74.689, -9.782]
  Set speed (500.0 mm/s)
  MoveL 438 to (139.15, 312.08, 6) mm, rotated rx 180 ry 0 rz 0 deg; joints [33.998, -56.771, 128.349, 35.569, -73.957, -10.321]
  MoveL 439 to (139.15, 131.49, 6) mm, rotated rx 180 ry 0 rz 0 deg; joints [26.326, -59.929, 135.434, 27.167, -76.171, -6.291]
  Set speed (25.4 mm/s)
  MoveL 440 to (139.15, 131.49, -3.54) mm, rotated rx -180 ry 0 rz 0 deg; joints [26.331, -59.213, 135.417, 27.096, -76.794, -5.964]
  MoveC 441 to (139.34, 131.49, -3.99) mm, rotated rx -180 ry 0 rz 0 deg; joints [26.335, -59.185, 135.429, 27.097, -76.83, -5.947] to (139.79, 131.48, -4.17) mm, rotated rx 180 ry 0 rz 0 deg; joints [26.346, -59.185, 135.459, 27.104, -76.858, -5.935]
  Set speed (50.8 mm/s)
  MoveL 442 to (140.42, 131.49, -4.18) mm, rotated rx -180 ry 0 rz 0 deg; joints [26.36, -59.205, 135.503, 27.116, -76.881, -5.926]
  MoveC 443 to (140.87, 131.3, -4.18) mm, rotated rx -180 ry 0 rz 0 deg; joints [26.362, -59.221, 135.54, 27.115, -76.9, -5.917] to (141.06, 130.85, -4.17) mm, rotated rx -180 ry 0 rz 0 deg; joints [26.345, -59.234, 135.568, 27.097, -76.912, -5.906]
  MoveL 444 to (141.06, 105.45, -4.18) mm, rotated rx -180 ry 0 rz 0 deg; joints [25.169, -59.59, 136.411, 25.847, -77.225, -5.433]
  MoveL 445 to (90.26, 105.45, -4.18) mm, rotated rx -180 ry 0 rz 0 deg; joints [24.097, -57.984, 132.859, 24.953, -75.356, -6.048]
  MoveL 446 to (90.26, 156.25, -4.18) mm, rotated rx 180 ry 0 rz 0 deg; joints [26.356, -57.256, 131.174, 27.387, -74.765, -7.05]
  MoveL 447 to (141.06, 156.25, -4.18) mm, rotated rx 180 ry 0 rz 0 deg; joints [27.499, -58.858, 134.686, 28.33, -76.593, -6.4]
  MoveL 448 to (141.06, 130.85, -4.17) mm, rotated rx -180 ry 0 rz 0 deg; joints [26.345, -59.234, 135.568, 27.097, -76.912, -5.906]
  MoveC 449 to (140.87, 130.4, -4.18) mm, rotated rx -180 ry 0 rz 0 deg; joints [26.321, -59.234, 135.57, 27.072, -76.911, -5.9] to (140.42, 130.21, -4.18) mm, rotated rx 180 ry 0 rz 0 deg; joints [26.302, -59.223, 135.546, 27.054, -76.897, -5.902]
  MoveL 450 to (139.79, 130.22, -4.18) mm, rotated rx -180 ry 0 rz 0 deg; joints [26.288, -59.203, 135.502, 27.042, -76.874, -5.91]
  MoveC 451 to (139.34, 130.21, -3.99) mm, rotated rx -180 ry 0 rz 0 deg; joints [26.277, -59.204, 135.472, 27.034, -76.846, -5.922] to (139.15, 130.22, -3.54) mm, rotated rx -180 ry 0 rz 0 deg; joints [26.273, -59.232, 135.46, 27.034, -76.81, -5.94]
  Set speed (500.0 mm/s)
  MoveL 452 to (139.15, 130.21, 5) mm, rotated rx 180 ry 0 rz 0 deg; joints [26.268, -59.873, 135.476, 27.097, -76.252, -6.232]
  MoveL 453 to (139.15, 131.48, 5) mm, rotated rx -180 ry 0 rz 0 deg; joints [26.326, -59.854, 135.432, 27.16, -76.237, -6.256]
  Set speed (25.4 mm/s)
  MoveL 454 to (139.15, 131.48, 1.82) mm, rotated rx 180 ry 0 rz 0 deg; joints [26.328, -59.616, 135.427, 27.136, -76.444, -6.147]
  MoveL 455 to (139.15, 131.48, -7.72) mm, rotated rx 180 ry 0 rz 0 deg; joints [26.333, -58.899, 135.407, 27.066, -77.065, -5.823]
  MoveC 456 to (139.34, 131.49, -8.16) mm, rotated rx -180 ry 0 rz 0 deg; joints [26.338, -58.871, 135.418, 27.067, -77.101, -5.805] to (139.79, 131.49, -8.35) mm, rotated rx 180 ry 0 rz 0 deg; joints [26.348, -58.87, 135.448, 27.074, -77.129, -5.793]
  Set speed (50.8 mm/s)
  MoveL 457 to (140.42, 131.49, -8.35) mm, rotated rx -180 ry 0 rz 0 deg; joints [26.363, -58.89, 135.492, 27.086, -77.152, -5.785]
  MoveC 458 to (140.87, 131.3, -8.35) mm, rotated rx -180 ry 0 rz 0 deg; joints [26.364, -58.906, 135.529, 27.086, -77.171, -5.775] to (141.06, 130.85, -8.35) mm, rotated rx 180 ry 0 rz 0 deg; joints [26.348, -58.918, 135.557, 27.068, -77.184, -5.764]
  MoveL 459 to (141.06, 105.45, -8.35) mm, rotated rx -180 ry 0 rz 0 deg; joints [25.171, -59.27, 136.4, 25.819, -77.504, -5.295]
  MoveL 460 to (90.26, 105.45, -8.35) mm, rotated rx -180 ry 0 rz 0 deg; joints [24.099, -57.682, 132.848, 24.923, -75.62, -5.922]
  MoveL 461 to (90.26, 156.25, -8.35) mm, rotated rx 180 ry 0 rz 0 deg; joints [26.359, -56.963, 131.164, 27.354, -75.017, -6.915]
  MoveL 462 to (141.06, 156.25, -8.35) mm, rotated rx -180 ry 0 rz 0 deg; joints [27.501, -58.547, 134.676, 28.299, -76.857, -6.255]
  MoveL 463 to (141.06, 130.85, -8.35) mm, rotated rx 180 ry 0 rz 0 deg; joints [26.348, -58.918, 135.557, 27.068, -77.184, -5.764]
  MoveC 464 to (140.87, 130.4, -8.35) mm, rotated rx -180 ry 0 rz 0 deg; joints [26.323, -58.919, 135.56, 27.042, -77.182, -5.758] to (140.42, 130.21, -8.35) mm, rotated rx -180 ry 0 rz 0 deg; joints [26.304, -58.908, 135.535, 27.024, -77.169, -5.761]
  MoveL 465 to (139.79, 130.22, -8.35) mm, rotated rx -180 ry 0 rz 0 deg; joints [26.29, -58.888, 135.492, 27.012, -77.146, -5.769]
  MoveC 466 to (139.34, 130.21, -8.16) mm, rotated rx 180 ry 0 rz 0 deg; joints [26.28, -58.889, 135.461, 27.005, -77.117, -5.781] to (139.15, 130.21, -7.72) mm, rotated rx -180 ry 0 rz 0 deg; joints [26.275, -58.917, 135.45, 27.004, -77.081, -5.798]
  Set speed (500.0 mm/s)
  MoveL 467 to (139.15, 130.21, 6) mm, rotated rx 180 ry 0 rz 0 deg; joints [26.267, -59.948, 135.477, 27.105, -76.186, -6.266]
  MoveL 468 to (266.15, 131.48, 6) mm, rotated rx 180 ry 0 rz 0 deg; joints [29.524, -63.804, 143.886, 29.967, -80.514, -4.663]
  Set speed (25.4 mm/s)
  MoveL 469 to (266.15, 131.49, -3.54) mm, rotated rx -180 ry 0 rz 0 deg; joints [29.53, -62.966, 143.867, 29.907, -81.224, -4.251]
  MoveC 470 to (266.34, 131.49, -3.99) mm, rotated rx -180 ry 0 rz 0 deg; joints [29.536, -62.932, 143.878, 29.909, -81.263, -4.229] to (266.79, 131.48, -4.17) mm, rotated rx -180 ry 0 rz 0 deg; joints [29.548, -62.928, 143.906, 29.92, -81.292, -4.214]
  Set speed (50.8 mm/s)
  MoveL 471 to (267.42, 131.49, -4.18) mm, rotated rx 180 ry 0 rz 0 deg; joints [29.566, -62.946, 143.947, 29.936, -81.314, -4.205]
  MoveC 472 to (267.87, 131.3, -4.17) mm, rotated rx 180 ry 0 rz 0 deg; joints [29.569, -62.961, 143.983, 29.938, -81.332, -4.195] to (268.06, 130.85, -4.17) mm, rotated rx -180 ry 0 rz 0 deg; joints [29.552, -62.973, 144.011, 29.919, -81.345, -4.184]
  MoveL 473 to (268.06, 105.45, -4.18) mm, rotated rx 180 ry 0 rz 0 deg; joints [28.28, -63.334, 144.917, 28.597, -81.726, -3.746]
  MoveL 474 to (217.26, 105.45, -4.18) mm, rotated rx -180 ry 0 rz 0 deg; joints [26.954, -61.885, 141.577, 27.401, -79.956, -4.452]
  MoveL 475 to (217.26, 156.25, -4.17) mm, rotated rx -180 ry 0 rz 0 deg; joints [29.393, -61.146, 139.781, 29.964, -79.249, -5.376]
  MoveL 476 to (268.06, 156.25, -4.18) mm, rotated rx -180 ry 0 rz 0 deg; joints [30.794, -62.592, 143.066, 31.216, -80.96, -4.648]
  MoveL 477 to (268.06, 130.85, -4.17) mm, rotated rx -180 ry 0 rz 0 deg; joints [29.552, -62.973, 144.011, 29.919, -81.345, -4.184]
  MoveC 478 to (267.87, 130.4, -4.17) mm, rotated rx -180 ry 0 rz 0 deg; joints [29.525, -62.974, 144.016, 29.891, -81.345, -4.179] to (267.42, 130.21, -4.18) mm, rotated rx -180 ry 0 rz 0 deg; joints [29.503, -62.965, 143.994, 29.87, -81.333, -4.182]
  MoveL 479 to (266.79, 130.21, -4.17) mm, rotated rx -180 ry 0 rz 0 deg; joints [29.485, -62.947, 143.953, 29.854, -81.311, -4.192]
  MoveC 480 to (266.34, 130.21, -3.99) mm, rotated rx -180 ry 0 rz 0 deg; joints [29.473, -62.951, 143.924, 29.844, -81.282, -4.206] to (266.15, 130.21, -3.54) mm, rotated rx -180 ry 0 rz 0 deg; joints [29.467, -62.985, 143.913, 29.842, -81.243, -4.228]
  Set speed (500.0 mm/s)
  MoveL 481 to (266.15, 130.21, 5) mm, rotated rx -180 ry 0 rz 0 deg; joints [29.462, -63.735, 143.931, 29.894, -80.607, -4.597]
  MoveL 482 to (266.15, 131.49, 5) mm, rotated rx 180 ry 0 rz 0 deg; joints [29.524, -63.716, 143.885, 29.96, -80.589, -4.62]
  Set speed (25.4 mm/s)
  MoveL 483 to (266.15, 131.48, 1.83) mm, rotated rx -180 ry 0 rz 0 deg; joints [29.526, -63.438, 143.879, 29.94, -80.825, -4.482]
  MoveL 484 to (266.15, 131.48, -7.71) mm, rotated rx 180 ry 0 rz 0 deg; joints [29.533, -62.599, 143.856, 29.883, -81.533, -4.072]
  MoveC 485 to (266.34, 131.48, -8.16) mm, rotated rx -180 ry 0 rz 0 deg; joints [29.538, -62.564, 143.866, 29.885, -81.572, -4.05] to (266.79, 131.49, -8.35) mm, rotated rx -180 ry 0 rz 0 deg; joints [29.551, -62.56, 143.895, 29.896, -81.601, -4.035]
  Set speed (50.8 mm/s)
  MoveL 486 to (267.42, 131.49, -8.35) mm, rotated rx -180 ry 0 rz 0 deg; joints [29.569, -62.578, 143.935, 29.912, -81.623, -4.025]
  MoveC 487 to (267.87, 131.3, -8.35) mm, rotated rx 180 ry 0 rz 0 deg; joints [29.572, -62.593, 143.971, 29.914, -81.641, -4.015] to (268.06, 130.85, -8.35) mm, rotated rx 180 ry 0 rz 0 deg; joints [29.555, -62.604, 144, 29.896, -81.654, -4.005]
  MoveL 488 to (268.06, 105.45, -8.35) mm, rotated rx 180 ry 0 rz 0 deg; joints [28.283, -62.959, 144.905, 28.575, -82.046, -3.57]
  MoveL 489 to (217.26, 105.45, -8.35) mm, rotated rx -180 ry 0 rz 0 deg; joints [26.957, -61.533, 141.566, 27.376, -80.258, -4.293]
  MoveL 490 to (217.26, 156.25, -8.35) mm, rotated rx -180 ry 0 rz 0 deg; joints [29.396, -60.806, 139.77, 29.936, -79.534, -5.21]
  MoveL 491 to (268.06, 156.25, -8.35) mm, rotated rx -180 ry 0 rz 0 deg; joints [30.796, -62.23, 143.055, 31.19, -81.26, -4.465]
  MoveL 492 to (268.06, 130.85, -8.35) mm, rotated rx -180 ry 0 rz 0 deg; joints [29.555, -62.604, 144, 29.896, -81.654, -4.005]
  MoveC 493 to (267.87, 130.4, -8.35) mm, rotated rx -180 ry 0 rz 0 deg; joints [29.528, -62.606, 144.004, 29.868, -81.655, -4] to (267.42, 130.21, -8.35) mm, rotated rx 180 ry 0 rz 0 deg; joints [29.506, -62.596, 143.982, 29.847, -81.642, -4.003]
  MoveL 494 to (266.79, 130.22, -8.35) mm, rotated rx -180 ry 0 rz 0 deg; joints [29.488, -62.579, 143.941, 29.83, -81.621, -4.013]
  MoveC 495 to (266.34, 130.21, -8.16) mm, rotated rx 180 ry 0 rz 0 deg; joints [29.475, -62.583, 143.913, 29.82, -81.592, -4.027] to (266.15, 130.22, -7.72) mm, rotated rx 180 ry 0 rz 0 deg; joints [29.47, -62.617, 143.902, 29.818, -81.552, -4.049]
  Set speed (500.0 mm/s)
  MoveL 496 to (266.15, 130.21, 6) mm, rotated rx -180 ry 0 rz 0 deg; joints [29.461, -63.823, 143.932, 29.901, -80.532, -4.64]
  MoveL 497 to (393.15, 131.48, 6) mm, rotated rx 180 ry 0 rz 0 deg; joints [33.506, -67.301, 151.798, 33.67, -84.545, -2.775]
  Set speed (25.4 mm/s)
  MoveL 498 to (393.15, 131.48, -3.54) mm, rotated rx -180 ry 0 rz 0 deg; joints [33.513, -66.301, 151.777, 33.63, -85.361, -2.232]
  MoveC 499 to (393.34, 131.49, -3.99) mm, rotated rx -180 ry 0 rz 0 deg; joints [33.52, -66.258, 151.787, 33.634, -85.405, -2.203] to (393.79, 131.48, -4.17) mm, rotated rx 180 ry 0 rz 0 deg; joints [33.536, -66.249, 151.813, 33.649, -85.435, -2.184]
  Set speed (50.8 mm/s)
  MoveL 500 to (394.42, 131.49, -4.17) mm, rotated rx -180 ry 0 rz 0 deg; joints [33.559, -66.265, 151.851, 33.67, -85.454, -2.173]
  MoveC 501 to (394.87, 131.3, -4.17) mm, rotated rx 180 ry 0 rz 0 deg; joints [33.564, -66.278, 151.886, 33.675, -85.472, -2.162] to (395.06, 130.85, -4.17) mm, rotated rx -180 ry 0 rz 0 deg; joints [33.547, -66.289, 151.915, 33.657, -85.486, -2.151]
  MoveL 502 to (395.06, 105.45, -4.17) mm, rotated rx -180 ry 0 rz 0 deg; joints [32.177, -66.647, 152.905, 32.258, -85.964, -1.724]
  MoveL 503 to (344.26, 105.45, -4.18) mm, rotated rx 180 ry 0 rz 0 deg; joints [30.508, -65.379, 149.773, 30.667, -84.303, -2.584]
  MoveL 504 to (344.26, 156.25, -4.17) mm, rotated rx -180 ry 0 rz 0 deg; joints [33.133, -64.636, 147.826, 33.372, -83.433, -3.468]
  MoveL 505 to (395.06, 156.25, -4.18) mm, rotated rx 180 ry 0 rz 0 deg; joints [34.875, -65.91, 150.885, 35.019, -85.011, -2.609]
  MoveL 506 to (395.06, 130.85, -4.17) mm, rotated rx -180 ry 0 rz 0 deg; joints [33.547, -66.289, 151.915, 33.657, -85.486, -2.151]
  MoveC 507 to (394.87, 130.4, -4.18) mm, rotated rx -180 ry 0 rz 0 deg; joints [33.517, -66.291, 151.921, 33.626, -85.489, -2.146] to (394.42, 130.22, -4.17) mm, rotated rx -180 ry 0 rz 0 deg; joints [33.491, -66.283, 151.902, 33.601, -85.478, -2.151]
  MoveL 508 to (393.79, 130.21, -4.18) mm, rotated rx -180 ry 0 rz 0 deg; joints [33.469, -66.268, 151.863, 33.58, -85.458, -2.162]
  MoveC 509 to (393.34, 130.21, -3.99) mm, rotated rx 180 ry 0 rz 0 deg; joints [33.453, -66.276, 151.837, 33.565, -85.428, -2.181] to (393.15, 130.22, -3.54) mm, rotated rx 180 ry 0 rz 0 deg; joints [33.446, -66.319, 151.827, 33.561, -85.384, -2.209]
  Set speed (500.0 mm/s)
  MoveL 510 to (393.15, 130.21, 5) mm, rotated rx -180 ry 0 rz 0 deg; joints [33.439, -67.216, 151.847, 33.596, -84.653, -2.696]
  MoveL 511 to (393.15, 131.49, 5) mm, rotated rx -180 ry 0 rz 0 deg; joints [33.507, -67.196, 151.797, 33.665, -84.631, -2.718]
  Set speed (25.4 mm/s)
  MoveL 512 to (393.15, 131.48, 1.82) mm, rotated rx 180 ry 0 rz 0 deg; joints [33.509, -66.864, 151.79, 33.651, -84.903, -2.537]
  MoveL 513 to (393.15, 131.49, -7.72) mm, rotated rx -180 ry 0 rz 0 deg; joints [33.517, -65.861, 151.764, 33.615, -85.715, -1.995]
  MoveC 514 to (393.34, 131.49, -8.16) mm, rotated rx 180 ry 0 rz 0 deg; joints [33.524, -65.819, 151.773, 33.619, -85.759, -1.966] to (393.79, 131.48, -8.35) mm, rotated rx 180 ry 0 rz 0 deg; joints [33.539, -65.81, 151.799, 33.634, -85.789, -1.948]
  Set speed (50.8 mm/s)
  MoveL 515 to (394.42, 131.48, -8.35) mm, rotated rx 180 ry 0 rz 0 deg; joints [33.562, -65.825, 151.838, 33.655, -85.809, -1.936]
  MoveC 516 to (394.87, 131.3, -8.35) mm, rotated rx -180 ry 0 rz 0 deg; joints [33.568, -65.838, 151.872, 33.66, -85.827, -1.925] to (395.06, 130.85, -8.35) mm, rotated rx -180 ry 0 rz 0 deg; joints [33.55, -65.848, 151.901, 33.642, -85.842, -1.914]
  MoveL 517 to (395.06, 105.45, -8.35) mm, rotated rx -180 ry 0 rz 0 deg; joints [32.18, -66.195, 152.891, 32.246, -86.335, -1.49]
  MoveL 518 to (344.26, 105.45, -8.35) mm, rotated rx 180 ry 0 rz 0 deg; joints [30.511, -64.96, 149.76, 30.65, -84.652, -2.377]
  MoveL 519 to (344.26, 156.25, -8.35) mm, rotated rx -180 ry 0 rz 0 deg; joints [33.137, -64.236, 147.813, 33.351, -83.757, -3.254]
  MoveL 520 to (395.06, 156.25, -8.35) mm, rotated rx -180 ry 0 rz 0 deg; joints [34.879, -65.48, 150.872, 35.002, -85.352, -2.369]
  MoveL 521 to (395.06, 130.85, -8.35) mm, rotated rx -180 ry 0 rz 0 deg; joints [33.55, -65.848, 151.901, 33.642, -85.842, -1.914]
  MoveC 522 to (394.87, 130.4, -8.35) mm, rotated rx -180 ry 0 rz 0 deg; joints [33.52, -65.85, 151.908, 33.612, -85.845, -1.909] to (394.42, 130.22, -8.35) mm, rotated rx -180 ry 0 rz 0 deg; joints [33.494, -65.842, 151.888, 33.586, -85.834, -1.914]
  MoveL 523 to (393.79, 130.22, -8.35) mm, rotated rx -180 ry 0 rz 0 deg; joints [33.472, -65.827, 151.85, 33.565, -85.814, -1.926]
  MoveC 524 to (393.34, 130.22, -8.16) mm, rotated rx 180 ry 0 rz 0 deg; joints [33.456, -65.836, 151.824, 33.55, -85.784, -1.944] to (393.15, 130.21, -7.72) mm, rotated rx -180 ry 0 rz 0 deg; joints [33.449, -65.879, 151.814, 33.546, -85.74, -1.973]
  Set speed (500.0 mm/s)
  MoveL 525 to (393.15, 130.22, 6) mm, rotated rx -180 ry 0 rz 0 deg; joints [33.438, -67.321, 151.849, 33.601, -84.567, -2.753]
  MoveL 526 to (393.15, -54.85, 6) mm, rotated rx -180 ry 0 rz 30 deg; joints [30.961, -66.473, 149.956, 61.206, -85.957, -5.908]
  Set speed (25.4 mm/s)
  MoveL 527 to (393.15, -54.85, -3.54) mm, rotated rx -180 ry 0 rz 30 deg; joints [30.968, -65.516, 149.935, 61.158, -86.409, -5.086]
  MoveC 528 to (393.34, -54.85, -3.99) mm, rotated rx -180 ry 0 rz 30 deg; joints [30.974, -65.476, 149.945, 61.162, -86.434, -5.042] to (393.79, -54.85, -4.17) mm, rotated rx 180 ry 0 rz 30 deg; joints [30.988, -65.468, 149.973, 61.174, -86.452, -5.013]
  Set speed (50.8 mm/s)
  MoveL 529 to (394.42, -54.85, -4.17) mm, rotated rx -180 ry 0 rz 30 deg; joints [31.008, -65.485, 150.012, 61.193, -86.465, -4.993]
  MoveC 530 to (394.87, -55.04, -4.17) mm, rotated rx -180 ry 0 rz 30 deg; joints [31.013, -65.499, 150.047, 61.197, -86.475, -4.975] to (395.06, -55.49, -4.17) mm, rotated rx -180 ry 0 rz 30 deg; joints [30.995, -65.51, 150.075, 61.178, -86.482, -4.959]
  MoveL 531 to (395.06, -80.89, -4.18) mm, rotated rx -180 ry 0 rz 30 deg; joints [29.626, -65.853, 151.002, 59.781, -86.662, -4.39]
  MoveL 532 to (344.26, -80.89, -4.18) mm, rotated rx -180 ry 0 rz 0 deg; joints [19.611, -67.38, 155.465, 19.627, -87.326, -0.371]
  MoveL 533 to (344.26, -30.09, -4.17) mm, rotated rx -180 ry 0 rz 0 deg; joints [22.773, -66.947, 154.155, 22.809, -86.556, -0.81]
  MoveL 534 to (395.06, -30.09, -4.17) mm, rotated rx -180 ry 0 rz 0 deg; joints [24.145, -68.178, 157.475, 24.147, -88.489, -0.015]
  MoveL 535 to (395.06, -55.49, -4.18) mm, rotated rx 180 ry 0 rz 30 deg; joints [30.995, -65.51, 150.075, 61.178, -86.482, -4.959]
  MoveC 536 to (394.87, -55.94, -4.17) mm, rotated rx -180 ry 0 rz 30 deg; joints [30.965, -65.511, 150.08, 61.148, -86.481, -4.954] to (394.42, -56.12, -4.18) mm, rotated rx -180 ry 0 rz 30 deg; joints [30.941, -65.502, 150.059, 61.124, -86.473, -4.964]
  MoveL 537 to (393.79, -56.12, -4.18) mm, rotated rx -180 ry 0 rz 30 deg; joints [30.921, -65.486, 150.02, 61.105, -86.46, -4.983]
  MoveC 538 to (393.34, -56.12, -3.99) mm, rotated rx -180 ry 0 rz 30 deg; joints [30.906, -65.493, 149.993, 61.093, -86.442, -5.013] to (393.15, -56.12, -3.54) mm, rotated rx -180 ry 0 rz 30 deg; joints [30.9, -65.534, 149.982, 61.089, -86.417, -5.057]
  Set speed (500.0 mm/s)
  MoveL 539 to (393.15, -56.12, 5) mm, rotated rx -180 ry 0 rz 30 deg; joints [30.894, -66.391, 150.002, 61.132, -86.012, -5.792]
  MoveL 540 to (393.15, -54.85, 5) mm, rotated rx -180 ry 0 rz 30 deg; joints [30.961, -66.372, 149.954, 61.201, -86.005, -5.821]
  Set speed (25.4 mm/s)
  MoveL 541 to (393.15, -54.85, 1.83) mm, rotated rx -180 ry 0 rz 30 deg; joints [30.964, -66.054, 149.948, 61.184, -86.155, -5.547]
  MoveL 542 to (393.15, -54.85, -7.71) mm, rotated rx -180 ry 0 rz 30 deg; joints [30.971, -65.096, 149.922, 61.14, -86.606, -4.729]
  MoveC 543 to (393.34, -54.85, -8.16) mm, rotated rx 180 ry 0 rz 30 deg; joints [30.977, -65.055, 149.932, 61.143, -86.63, -4.685] to (393.79, -54.85, -8.35) mm, rotated rx -180 ry 0 rz 30 deg; joints [30.991, -65.048, 149.959, 61.156, -86.648, -4.655]
  Set speed (50.8 mm/s)
  MoveL 544 to (394.42, -54.85, -8.35) mm, rotated rx -180 ry 0 rz 30 deg; joints [31.012, -65.064, 149.999, 61.175, -86.661, -4.635]
  MoveC 545 to (394.87, -55.04, -8.35) mm, rotated rx -180 ry 0 rz 30 deg; joints [31.016, -65.077, 150.034, 61.178, -86.672, -4.617] to (395.06, -55.49, -8.35) mm, rotated rx -180 ry 0 rz 30 deg; joints [30.998, -65.088, 150.062, 61.159, -86.679, -4.601]
  MoveL 546 to (395.06, -80.89, -8.35) mm, rotated rx -180 ry 0 rz 30 deg; joints [29.629, -65.422, 150.988, 59.763, -86.873, -4.029]
  MoveL 547 to (344.26, -80.89, -8.35) mm, rotated rx -180 ry 0 rz 0 deg; joints [19.614, -66.896, 155.449, 19.623, -87.768, -0.213]
  MoveL 548 to (344.26, -30.09, -8.35) mm, rotated rx -180 ry 0 rz 0 deg; joints [22.776, -66.48, 154.14, 22.802, -86.973, -0.635]
  MoveL 549 to (395.06, -30.09, -8.35) mm, rotated rx -180 ry 0 rz 0 deg; joints [24.148, -67.665, 157.459, 24.145, -88.942, 0.188]
  MoveL 550 to (395.06, -55.49, -8.35) mm, rotated rx -180 ry 0 rz 30 deg; joints [30.998, -65.088, 150.062, 61.159, -86.679, -4.601]
  MoveC 551 to (394.87, -55.94, -8.35) mm, rotated rx -180 ry 0 rz 30 deg; joints [30.968, -65.09, 150.067, 61.129, -86.678, -4.596] to (394.42, -56.12, -8.35) mm, rotated rx -180 ry 0 rz 30 deg; joints [30.944, -65.081, 150.046, 61.106, -86.671, -4.606]
  MoveL 552 to (393.79, -56.12, -8.35) mm, rotated rx -180 ry 0 rz 30 deg; joints [30.924, -65.065, 150.007, 61.087, -86.658, -4.626]
  MoveC 553 to (393.34, -56.12, -8.16) mm, rotated rx -180 ry 0 rz 30 deg; joints [30.909, -65.073, 149.979, 61.074, -86.64, -4.656] to (393.15, -56.12, -7.72) mm, rotated rx 180 ry 0 rz 30 deg; joints [30.903, -65.113, 149.969, 61.071, -86.615, -4.7]
  Set speed (500.0 mm/s)
  MoveL 554 to (393.15, -56.12, 6) mm, rotated rx -180 ry 0 rz 30 deg; joints [30.893, -66.491, 150.003, 61.137, -85.964, -5.879]
  MoveL 555 to (266.15, -54.85, 6) mm, rotated rx -180 ry 0 rz 0 deg; joints [19.502, -66.111, 149.57, 19.649, -82.967, -1.923]
  Set speed (25.4 mm/s)
  MoveL 556 to (266.15, -54.85, -3.54) mm, rotated rx -180 ry 0 rz 0 deg; joints [19.507, -65.162, 149.548, 19.619, -83.84, -1.61]
  MoveC 557 to (266.34, -54.85, -3.99) mm, rotated rx 180 ry 0 rz 0 deg; joints [19.511, -65.123, 149.56, 19.621, -83.888, -1.593] to (266.79, -54.85, -4.17) mm, rotated rx 180 ry 0 rz 0 deg; joints [19.521, -65.117, 149.59, 19.629, -83.922, -1.582]
  Set speed (50.8 mm/s)
  MoveL 558 to (267.42, -54.85, -4.18) mm, rotated rx 180 ry 0 rz 0 deg; joints [19.534, -65.134, 149.633, 19.641, -83.947, -1.574]
  MoveC 559 to (267.87, -55.04, -4.18) mm, rotated rx 180 ry 0 rz 0 deg; joints [19.532, -65.148, 149.668, 19.639, -83.967, -1.567] to (268.06, -55.49, -4.18) mm, rotated rx 180 ry 0 rz 0 deg; joints [19.51, -65.158, 149.692, 19.616, -83.98, -1.56]
  MoveL 560 to (268.06, -80.89, -4.18) mm, rotated rx 180 ry 0 rz 0 deg; joints [18.021, -65.371, 150.283, 18.107, -84.293, -1.307]
  MoveL 561 to (217.26, -80.89, -4.18) mm, rotated rx -180 ry 0 rz 0 deg; joints [17.093, -63.925, 146.756, 17.248, -82.28, -1.848]
  MoveL 562 to (217.26, -30.09, -4.18) mm, rotated rx -180 ry 0 rz 0 deg; joints [19.916, -63.474, 145.574, 20.128, -81.707, -2.439]
  MoveL 563 to (268.06, -30.09, -4.17) mm, rotated rx 180 ry 0 rz 0 deg; joints [20.972, -64.924, 149.055, 21.101, -83.652, -1.838]
  MoveL 564 to (268.06, -55.49, -4.18) mm, rotated rx 180 ry 0 rz 0 deg; joints [19.51, -65.158, 149.692, 19.616, -83.98, -1.56]
  MoveC 565 to (267.87, -55.94, -4.18) mm, rotated rx 180 ry 0 rz 0 deg; joints [19.48, -65.156, 149.69, 19.586, -83.978, -1.558] to (267.42, -56.12, -4.17) mm, rotated rx 180 ry 0 rz 0 deg; joints [19.46, -65.146, 149.664, 19.566, -83.963, -1.561]
  MoveL 566 to (266.79, -56.12, -4.18) mm, rotated rx 180 ry 0 rz 0 deg; joints [19.447, -65.128, 149.62, 19.554, -83.938, -1.569]
  MoveC 567 to (266.34, -56.12, -3.99) mm, rotated rx -180 ry 0 rz 0 deg; joints [19.438, -65.134, 149.59, 19.546, -83.904, -1.58] to (266.15, -56.12, -3.54) mm, rotated rx 180 ry 0 rz 0 deg; joints [19.434, -65.174, 149.579, 19.544, -83.856, -1.597]
  Set speed (500.0 mm/s)
  MoveL 568 to (266.15, -56.12, 5) mm, rotated rx -180 ry 0 rz 0 deg; joints [19.429, -66.023, 149.599, 19.571, -83.074, -1.876]
  MoveL 569 to (266.15, -54.85, 5) mm, rotated rx 180 ry 0 rz 0 deg; joints [19.502, -66.011, 149.568, 19.646, -83.059, -1.89]
  Set speed (25.4 mm/s)
  MoveL 570 to (266.15, -54.85, 1.83) mm, rotated rx -180 ry 0 rz 0 deg; joints [19.504, -65.696, 149.562, 19.635, -83.35, -1.786]
  MoveL 571 to (266.15, -54.85, -7.71) mm, rotated rx -180 ry 0 rz 0 deg; joints [19.51, -64.746, 149.535, 19.607, -84.22, -1.474]
  MoveC 572 to (266.34, -54.85, -8.16) mm, rotated rx -180 ry 0 rz 0 deg; joints [19.514, -64.706, 149.546, 19.609, -84.268, -1.458] to (266.79, -54.85, -8.35) mm, rotated rx -180 ry 0 rz 0 deg; joints [19.523, -64.7, 149.576, 19.617, -84.302, -1.446]
  Set speed (50.8 mm/s)
  MoveL 573 to (267.42, -54.85, -8.35) mm, rotated rx -180 ry 0 rz 0 deg; joints [19.536, -64.717, 149.62, 19.63, -84.327, -1.438]
